C09145=1170.053,255.374,-66.162,-177.310,7.479,148.636
C09146=1170.048,255.622,-66.190,-177.307,7.482,148.635
C09147=1170.043,255.871,-66.218,-177.305,7.485,148.635
C09148=1170.039,256.120,-66.245,-177.302,7.488,148.635
C09149=1170.034,256.368,-66.273,-177.300,7.490,148.635
C09150=1170.030,256.617,-66.300,-177.297,7.493,148.635
C09151=1170.025,256.865,-66.328,-177.294,7.496,148.635
C09152=1170.021,257.114,-66.355,-177.291,7.499,148.635
C09153=1170.017,257.362,-66.383,-177.289,7.501,148.635
C09154=1170.012,257.610,-66.410,-177.286,7.504,148.635
C09155=1170.009,257.859,-66.438,-177.283,7.507,148.635
C09156=1170.004,258.107,-66.465,-177.280,7.510,148.635
C09157=1170.000,258.355,-66.493,-177.278,7.512,148.634
C09158=1169.996,258.604,-66.521,-177.276,7.515,148.634
C09159=1169.991,258.852,-66.548,-177.273,7.518,148.634
C09160=1169.987,259.101,-66.575,-177.270,7.521,148.634
C09161=1169.982,259.350,-66.604,-177.267,7.523,148.634
C09162=1169.977,259.598,-66.631,-177.265,7.526,148.634
C09163=1169.973,259.846,-66.659,-177.262,7.529,148.634
C09164=1169.969,260.095,-66.686,-177.259,7.532,148.634
C09165=1169.965,260.343,-66.714,-177.257,7.534,148.634
C09166=1169.960,260.591,-66.742,-177.254,7.537,148.634
C09167=1169.955,260.840,-66.770,-177.251,7.540,148.634
C09168=1169.951,261.088,-66.798,-177.249,7.543,148.634
C09169=1169.947,261.337,-66.826,-177.246,7.545,148.633
C09170=1169.943,261.585,-66.853,-177.244,7.548,148.633
C09171=1169.938,261.859,-66.884,-177.241,7.551,148.633
C09172=1169.933,262.131,-66.914,-177.238,7.553,148.633
C09173=1169.928,262.405,-66.945,-177.234,7.557,148.633
C09174=1169.924,262.677,-66.976,-177.232,7.560,148.633
C09175=1169.919,262.926,-67.003,-177.230,7.562,148.633
C09176=1169.915,263.175,-67.032,-177.227,7.565,148.633
C09177=1169.910,263.423,-67.060,-177.224,7.568,148.633
C09178=1169.907,263.671,-67.088,-177.221,7.571,148.633
C09179=1169.902,263.920,-67.115,-177.219,7.574,148.633
C09180=1169.897,264.168,-67.143,-177.216,7.576,148.633
C09181=1169.893,264.416,-67.171,-177.214,7.579,148.633
C09182=1169.889,264.664,-67.199,-177.211,7.582,148.633
C09183=1169.884,264.913,-67.228,-177.208,7.585,148.632
C09184=1169.880,265.161,-67.256,-177.205,7.588,148.632
C09185=1169.876,265.410,-67.283,-177.203,7.590,148.632
C09186=1169.871,265.658,-67.311,-177.200,7.593,148.632
C09187=1169.867,265.907,-67.340,-177.198,7.596,148.632
C09188=1169.863,266.155,-67.367,-177.195,7.599,148.632
C09189=1169.858,266.404,-67.396,-177.193,7.601,148.632
C09190=1169.854,266.652,-67.424,-177.190,7.604,148.632
C09191=1169.849,266.901,-67.453,-177.187,7.607,148.632
C09192=1169.845,267.148,-67.480,-177.184,7.610,148.632
C09193=1169.841,267.397,-67.509,-177.182,7.613,148.632
C09194=1169.836,267.645,-67.537,-177.180,7.615,148.632
C09195=1169.832,267.894,-67.565,-177.177,7.618,148.632
C09196=1169.827,268.142,-67.593,-177.174,7.621,148.632
C09197=1169.824,268.390,-67.622,-177.171,7.624,148.632
C09198=1169.818,268.639,-67.650,-177.169,7.627,148.632
C09199=1169.815,268.887,-67.678,-177.166,7.630,148.632
C09200=1169.810,269.135,-67.706,-177.164,7.632,148.631
C09201=1169.806,269.384,-67.735,-177.161,7.635,148.631
C09202=1169.801,269.632,-67.763,-177.158,7.638,148.631
C09203=1169.797,269.881,-67.791,-177.155,7.641,148.631
C09204=1169.792,270.128,-67.820,-177.153,7.644,148.631
C09205=1169.788,270.377,-67.848,-177.150,7.646,148.631
C09206=1169.784,270.626,-67.877,-177.148,7.649,148.631
C09207=1169.780,270.874,-67.905,-177.145,7.652,148.631
C09208=1169.775,271.123,-67.934,-177.142,7.655,148.631
C09209=1169.771,271.370,-67.961,-177.139,7.658,148.631
C09210=1169.767,271.619,-67.991,-177.137,7.661,148.631
C09211=1169.762,271.867,-68.019,-177.135,7.663,148.631
C09212=1169.758,272.115,-68.047,-177.132,7.666,148.631
C09213=1169.754,272.364,-68.075,-177.129,7.669,148.631
C09214=1169.749,272.612,-68.104,-177.126,7.672,148.631
C09215=1169.745,272.861,-68.133,-177.124,7.675,148.631
C09216=1169.741,273.109,-68.161,-177.121,7.678,148.631
C09217=1169.736,273.357,-68.190,-177.119,7.680,148.631
C09218=1169.732,273.605,-68.219,-177.116,7.683,148.631
C09219=1169.727,273.853,-68.247,-177.113,7.686,148.630
C09220=1169.723,274.102,-68.276,-177.110,7.689,148.630
C09221=1169.719,274.350,-68.305,-177.108,7.692,148.630
C09222=1169.714,274.598,-68.333,-177.105,7.695,148.631
C09223=1169.710,274.847,-68.362,-177.103,7.698,148.630
C09224=1169.706,275.095,-68.391,-177.100,7.701,148.630
C09225=1169.701,275.343,-68.419,-177.098,7.703,148.630
C09226=1169.697,275.592,-68.448,-177.095,7.706,148.630
C09227=1169.693,275.840,-68.477,-177.092,7.709,148.630
C09228=1169.688,276.089,-68.505,-177.089,7.712,148.630
C09229=1169.684,276.337,-68.534,-177.087,7.715,148.630
C09230=1169.680,276.585,-68.563,-177.085,7.718,148.630
C09231=1169.676,276.834,-68.592,-177.082,7.720,148.630
C09232=1169.671,277.082,-68.620,-177.079,7.723,148.630
C09233=1169.667,277.330,-68.650,-177.076,7.726,148.630
C09234=1169.663,277.579,-68.678,-177.074,7.730,148.630
C09235=1169.658,277.826,-68.707,-177.071,7.733,148.630
C09236=1169.654,278.075,-68.736,-177.069,7.736,148.630
C09237=1169.650,278.323,-68.765,-177.066,7.739,148.630
C09238=1169.646,278.571,-68.794,-177.064,7.741,148.630
C09239=1169.641,278.820,-68.822,-177.061,7.744,148.630
C09240=1169.637,279.068,-68.852,-177.058,7.747,148.630
C09241=1169.633,279.317,-68.881,-177.055,7.750,148.630
C09242=1169.628,279.565,-68.910,-177.053,7.753,148.630
C09243=1169.624,279.812,-68.939,-177.050,7.756,148.630
C09244=1169.620,280.061,-68.967,-177.048,7.759,148.630
C09245=1169.616,280.309,-68.997,-177.045,7.762,148.630
C09246=1169.611,280.558,-69.026,-177.043,7.764,148.630
C09247=1169.607,280.807,-69.055,-177.040,7.767,148.630
C09248=1169.602,281.054,-69.084,-177.037,7.770,148.630
C09249=1169.598,281.302,-69.114,-177.034,7.773,148.630
C09250=1169.594,281.551,-69.142,-177.032,7.776,148.630
C09251=1169.590,281.799,-69.171,-177.029,7.779,148.630
C09252=1169.586,282.047,-69.201,-177.027,7.782,148.630
C09253=1169.581,282.295,-69.230,-177.024,7.785,148.630
C09254=1169.577,282.544,-69.258,-177.022,7.787,148.630
C09255=1169.572,282.792,-69.288,-177.019,7.790,148.630
C09256=1169.568,283.040,-69.317,-177.016,7.793,148.630
C09257=1169.564,283.289,-69.347,-177.014,7.797,148.630
C09258=1169.560,283.537,-69.376,-177.011,7.799,148.630
C09259=1169.555,283.785,-69.405,-177.008,7.802,148.630
C09260=1169.551,284.033,-69.434,-177.006,7.805,148.630
C09261=1169.546,284.282,-69.464,-177.003,7.808,148.630
C09262=1169.542,284.530,-69.493,-177.000,7.811,148.630
C09263=1169.538,284.778,-69.522,-176.998,7.815,148.630
C09264=1169.534,285.026,-69.552,-176.996,7.817,148.630
C09265=1169.530,285.275,-69.581,-176.993,7.820,148.630
C09266=1169.525,285.522,-69.610,-176.990,7.823,148.630
C09267=1169.521,285.771,-69.640,-176.988,7.826,148.630
C09268=1169.517,286.019,-69.669,-176.985,7.829,148.630
C09269=1169.512,286.267,-69.699,-176.983,7.832,148.630
C09270=1169.508,286.515,-69.728,-176.980,7.835,148.630
C09271=1169.504,286.764,-69.758,-176.977,7.838,148.630
C09272=1169.500,287.012,-69.787,-176.974,7.841,148.630
C09273=1169.496,287.260,-69.817,-176.972,7.844,148.630
C09274=1169.491,287.508,-69.846,-176.969,7.847,148.630
C09275=1169.486,287.783,-69.878,-176.967,7.850,148.630
C09276=1169.481,288.058,-69.912,-176.964,7.853,148.630
C09277=1169.476,288.333,-69.944,-176.960,7.857,148.630
C09278=1169.472,288.608,-69.977,-176.958,7.860,148.630
C09279=1169.468,288.856,-70.007,-176.955,7.863,148.630
C09280=1169.463,289.105,-70.036,-176.953,7.866,148.630
C09281=1169.459,289.353,-70.066,-176.950,7.869,148.630
C09282=1169.455,289.601,-70.095,-176.947,7.872,148.630
C09283=1169.451,289.849,-70.125,-176.944,7.875,148.630
C09284=1169.447,290.098,-70.154,-176.942,7.878,148.630
C09285=1169.442,290.346,-70.185,-176.939,7.881,148.630
C09286=1169.438,290.594,-70.214,-176.937,7.883,148.630
C09287=1169.434,290.842,-70.244,-176.935,7.886,148.630
C09288=1169.429,291.090,-70.273,-176.932,7.890,148.630
C09289=1169.426,291.338,-70.304,-176.929,7.893,148.630
C09290=1169.421,291.587,-70.334,-176.927,7.896,148.630
C09291=1169.416,291.835,-70.363,-176.924,7.899,148.630
C09292=1169.412,292.083,-70.392,-176.922,7.902,148.630
C09293=1169.408,292.331,-70.423,-176.919,7.905,148.630
C09294=1169.404,292.579,-70.453,-176.916,7.908,148.630
C09295=1169.399,292.828,-70.482,-176.913,7.911,148.630
C09296=1169.395,293.075,-70.512,-176.911,7.914,148.630
C09297=1169.391,293.324,-70.542,-176.908,7.917,148.630
C09298=1169.386,293.572,-70.572,-176.906,7.920,148.630
C09299=1169.382,293.820,-70.602,-176.903,7.923,148.630
C09300=1169.378,294.068,-70.631,-176.901,7.926,148.630
C09301=1169.374,294.316,-70.662,-176.898,7.929,148.630
C09302=1169.370,294.564,-70.692,-176.895,7.932,148.630
C09303=1169.365,294.813,-70.721,-176.893,7.936,148.630
C09304=1169.361,295.061,-70.752,-176.890,7.939,148.630
C09305=1169.357,295.310,-70.782,-176.887,7.942,148.630
C09306=1169.353,295.557,-70.812,-176.885,7.944,148.630
C09307=1169.348,295.806,-70.842,-176.883,7.947,148.630
C09308=1169.344,296.053,-70.872,-176.880,7.950,148.630
C09309=1169.340,296.302,-70.902,-176.878,7.953,148.630
C09310=1169.336,296.550,-70.932,-176.875,7.956,148.630
C09311=1169.331,296.798,-70.962,-176.872,7.959,148.630
C09312=1169.327,297.046,-70.993,-176.870,7.962,148.630
C09313=1169.323,297.293,-71.023,-176.867,7.965,148.630
C09314=1169.319,297.543,-71.053,-176.865,7.968,148.630
C09315=1169.315,297.790,-71.083,-176.862,7.971,148.630
C09316=1169.311,298.039,-71.113,-176.859,7.974,148.630
C09317=1169.306,298.287,-71.143,-176.857,7.978,148.631
C09318=1169.302,298.534,-71.174,-176.854,7.981,148.631
C09319=1169.297,298.783,-71.204,-176.851,7.984,148.631
C09320=1169.294,299.031,-71.234,-176.849,7.987,148.631
C09321=1169.289,299.279,-71.265,-176.846,7.990,148.631
C09322=1169.285,299.527,-71.294,-176.844,7.993,148.631
C09323=1169.281,299.775,-71.325,-176.841,7.996,148.631
C09324=1169.277,300.023,-71.355,-176.839,7.999,148.631
C09325=1169.272,300.272,-71.385,-176.836,8.002,148.631
C09326=1169.268,300.520,-71.416,-176.834,8.005,148.631
C09327=1169.264,300.768,-71.447,-176.831,8.008,148.631
C09328=1169.259,301.016,-71.478,-176.829,8.012,148.631
C09329=1169.255,301.264,-71.507,-176.826,8.015,148.631
C09330=1169.250,301.512,-71.538,-176.823,8.018,148.631
C09331=1169.247,301.760,-71.568,-176.821,8.021,148.631
C09332=1169.243,302.008,-71.599,-176.818,8.024,148.631
C09333=1169.238,302.256,-71.630,-176.815,8.027,148.631
C09334=1169.234,302.504,-71.660,-176.813,8.030,148.631
C09335=1169.230,302.753,-71.690,-176.810,8.033,148.631
C09336=1169.226,303.001,-71.721,-176.808,8.036,148.631
C09337=1169.221,303.249,-71.751,-176.805,8.039,148.632
C09338=1169.217,303.497,-71.782,-176.803,8.042,148.632
C09339=1169.213,303.745,-71.813,-176.800,8.046,148.632
C09340=1169.209,303.993,-71.843,-176.798,8.049,148.632
C09341=1169.204,304.241,-71.874,-176.795,8.052,148.632
C09342=1169.200,304.489,-71.904,-176.793,8.055,148.632
C09343=1169.196,304.737,-71.935,-176.790,8.058,148.632
C09344=1169.192,304.985,-71.966,-176.787,8.061,148.632
C09345=1169.187,305.233,-71.997,-176.785,8.064,148.632
C09346=1169.184,305.482,-72.027,-176.782,8.067,148.632
C09347=1169.179,305.730,-72.058,-176.780,8.070,148.632
C09348=1169.175,305.978,-72.089,-176.777,8.073,148.632
C09349=1169.171,306.225,-72.119,-176.774,8.076,148.632
C09350=1169.167,306.474,-72.150,-176.772,8.080,148.632
C09351=1169.162,306.722,-72.181,-176.769,8.083,148.632
C09352=1169.157,306.970,-72.212,-176.767,8.086,148.632
C09353=1169.153,307.218,-72.243,-176.764,8.089,148.632
C09354=1169.150,307.466,-72.273,-176.762,8.092,148.633
C09355=1169.145,307.714,-72.304,-176.759,8.095,148.633
C09356=1169.141,307.962,-72.336,-176.756,8.098,148.633
C09357=1169.137,308.210,-72.367,-176.754,8.102,148.633
C09358=1169.132,308.458,-72.397,-176.751,8.105,148.633
C09359=1169.129,308.706,-72.428,-176.749,8.108,148.633
C09360=1169.124,308.954,-72.459,-176.746,8.111,148.633
C09361=1169.120,309.203,-72.490,-176.744,8.114,148.633
C09362=1169.116,309.450,-72.521,-176.741,8.118,148.633
C09363=1169.111,309.698,-72.552,-176.738,8.121,148.633
C09364=1169.107,309.947,-72.583,-176.736,8.124,148.633
C09365=1169.103,310.195,-72.613,-176.733,8.127,148.633
C09366=1169.100,310.443,-72.645,-176.731,8.130,148.633
C09367=1169.095,310.691,-72.676,-176.728,8.133,148.633
C09368=1169.090,310.939,-72.707,-176.726,8.137,148.634
C09369=1169.087,311.187,-72.738,-176.723,8.140,148.634
C09370=1169.082,311.435,-72.769,-176.721,8.143,148.634
C09371=1169.078,311.683,-72.800,-176.718,8.146,148.634
C09372=1169.074,311.931,-72.832,-176.716,8.149,148.634
C09373=1169.069,312.179,-72.863,-176.713,8.152,148.634
C09374=1169.065,312.427,-72.894,-176.711,8.156,148.634
C09375=1169.061,312.674,-72.925,-176.708,8.159,148.634
C09376=1169.057,312.923,-72.956,-176.706,8.162,148.634
C09377=1169.052,313.170,-72.988,-176.703,8.165,148.634
C09378=1169.048,313.419,-73.019,-176.701,8.168,148.635
C09379=1169.044,313.696,-73.054,-176.697,8.172,148.635
C09380=1169.039,313.972,-73.089,-176.695,8.175,148.635
C09381=1169.034,314.250,-73.123,-176.692,8.179,148.635
C09382=1169.030,314.526,-73.158,-176.689,8.182,148.635
C09383=1169.026,314.774,-73.190,-176.687,8.185,148.635
C09384=1169.021,315.023,-73.221,-176.683,8.189,148.635
C09385=1169.017,315.271,-73.253,-176.681,8.192,148.635
C09386=1169.013,315.519,-73.284,-176.678,8.195,148.635
C09387=1169.009,315.767,-73.316,-176.676,8.199,148.635
C09388=1169.004,316.015,-73.346,-176.673,8.202,148.635
C09389=1169.001,316.263,-73.378,-176.671,8.205,148.636
C09390=1168.997,316.511,-73.410,-176.668,8.208,148.636
C09391=1168.992,316.759,-73.441,-176.666,8.211,148.636
C09392=1168.989,317.007,-73.473,-176.664,8.214,148.636
C09393=1168.984,317.255,-73.503,-176.661,8.217,148.636
C09394=1168.980,317.503,-73.535,-176.659,8.221,148.636
C09395=1168.976,317.750,-73.567,-176.656,8.224,148.636
C09396=1168.971,317.998,-73.599,-176.654,8.227,148.636
C09397=1168.967,318.246,-73.630,-176.650,8.231,148.636
C09398=1168.963,318.494,-73.662,-176.648,8.234,148.637
C09399=1168.959,318.743,-73.694,-176.645,8.237,148.636
C09400=1168.955,318.990,-73.724,-176.643,8.240,148.637
C09401=1168.951,319.239,-73.756,-176.641,8.244,148.637
C09402=1168.946,319.486,-73.788,-176.638,8.247,148.637
C09403=1168.942,319.734,-73.820,-176.636,8.250,148.637
C09404=1168.939,319.982,-73.852,-176.633,8.253,148.637
C09405=1168.934,320.230,-73.883,-176.631,8.256,148.637
C09406=1168.930,320.478,-73.915,-176.628,8.259,148.637
C09407=1168.925,320.726,-73.947,-176.626,8.263,148.637
C09408=1168.922,320.974,-73.979,-176.623,8.266,148.638
C09409=1168.918,321.222,-74.010,-176.620,8.270,148.638
C09410=1168.914,321.469,-74.042,-176.618,8.273,148.638
C09411=1168.909,321.718,-74.074,-176.615,8.276,148.638
C09412=1168.905,321.966,-74.106,-176.613,8.279,148.638
C09413=1168.901,322.214,-74.137,-176.611,8.282,148.638
C09414=1168.896,322.462,-74.169,-176.608,8.285,148.638
C09415=1168.893,322.710,-74.201,-176.606,8.289,148.638
C09416=1168.888,322.957,-74.233,-176.603,8.292,148.638
C09417=1168.885,323.205,-74.265,-176.601,8.295,148.639
C09418=1168.880,323.454,-74.297,-176.598,8.299,148.639
C09419=1168.876,323.701,-74.329,-176.595,8.302,148.639
C09420=1168.872,323.949,-74.360,-176.593,8.305,148.639
C09421=1168.868,324.198,-74.393,-176.590,8.309,148.639
C09422=1168.863,324.445,-74.424,-176.588,8.312,148.639
C09423=1168.860,324.693,-74.456,-176.585,8.315,148.639
C09424=1168.855,324.941,-74.489,-176.583,8.318,148.639
C09425=1168.852,325.189,-74.521,-176.580,8.321,148.640
C09426=1168.847,325.436,-74.553,-176.578,8.325,148.640
C09427=1168.843,325.684,-74.585,-176.575,8.328,148.640
C09428=1168.839,325.932,-74.617,-176.572,8.332,148.640
C09429=1168.835,326.181,-74.649,-176.570,8.335,148.640
C09430=1168.831,326.428,-74.681,-176.567,8.338,148.640
C09431=1168.826,326.676,-74.713,-176.565,8.341,148.640
C09432=1168.823,326.924,-74.746,-176.563,8.345,148.641
C09433=1168.818,327.172,-74.778,-176.560,8.348,148.641
C09434=1168.814,327.420,-74.810,-176.558,8.351,148.641
C09435=1168.810,327.668,-74.842,-176.555,8.355,148.641
C09436=1168.806,327.916,-74.874,-176.552,8.358,148.641
C09437=1168.802,328.164,-74.907,-176.550,8.361,148.641
C09438=1168.797,328.411,-74.939,-176.548,8.365,148.642
C09439=1168.793,328.659,-74.971,-176.545,8.368,148.642
C09440=1168.789,328.907,-75.003,-176.543,8.371,148.642
C09441=1168.785,329.155,-75.036,-176.540,8.374,148.642
C09442=1168.781,329.403,-75.068,-176.537,8.378,148.642
C09443=1168.776,329.651,-75.100,-176.535,8.381,148.642
C09444=1168.773,329.898,-75.133,-176.532,8.384,148.642
C09445=1168.769,330.147,-75.165,-176.530,8.388,148.643
C09446=1168.765,330.395,-75.197,-176.528,8.391,148.643
C09447=1168.761,330.642,-75.230,-176.525,8.394,148.643
C09448=1168.756,330.890,-75.262,-176.523,8.397,148.643
C09449=1168.752,331.137,-75.295,-176.520,8.401,148.643
C09450=1168.748,331.386,-75.327,-176.517,8.404,148.643
C09451=1168.744,331.633,-75.360,-176.515,8.408,148.643
C09452=1168.740,331.881,-75.392,-176.513,8.411,148.644
C09453=1168.736,332.130,-75.425,-176.510,8.414,148.644
C09454=1168.732,332.377,-75.457,-176.508,8.418,148.644
C09455=1168.727,332.625,-75.489,-176.505,8.421,148.644
C09456=1168.723,332.873,-75.522,-176.503,8.425,148.644
C09457=1168.719,333.121,-75.554,-176.500,8.428,148.644
C09458=1168.715,333.368,-75.587,-176.498,8.431,148.645
C09459=1168.711,333.616,-75.620,-176.495,8.434,148.645
C09460=1168.707,333.864,-75.652,-176.493,8.438,148.645
C09461=1168.703,334.112,-75.685,-176.490,8.442,148.645
C09462=1168.699,334.360,-75.718,-176.488,8.445,148.645
C09463=1168.695,334.608,-75.751,-176.486,8.448,148.646
C09464=1168.691,334.855,-75.783,-176.483,8.451,148.646
C09465=1168.686,335.103,-75.816,-176.480,8.455,148.646
C09466=1168.682,335.351,-75.849,-176.478,8.458,148.646
C09467=1168.678,335.599,-75.881,-176.475,8.462,148.646
C09468=1168.674,335.847,-75.914,-176.473,8.465,148.646
C09469=1168.670,336.094,-75.947,-176.470,8.468,148.646
C09470=1168.666,336.342,-75.980,-176.468,8.472,148.647
C09471=1168.661,336.590,-76.013,-176.466,8.475,148.647
C09472=1168.658,336.838,-76.045,-176.463,8.479,148.647
C09473=1168.654,337.086,-76.078,-176.461,8.482,148.647
C09474=1168.649,337.334,-76.111,-176.458,8.486,148.647
C09475=1168.645,337.582,-76.144,-176.456,8.489,148.647
C09476=1168.641,337.829,-76.177,-176.453,8.492,148.648
C09477=1168.638,338.077,-76.210,-176.451,8.495,148.648
C09478=1168.634,338.324,-76.243,-176.448,8.499,148.648
C09479=1168.629,338.573,-76.275,-176.446,8.503,148.648
C09480=1168.625,338.821,-76.308,-176.444,8.506,148.649
C09481=1168.621,339.068,-76.342,-176.441,8.509,148.649
C09482=1168.617,339.316,-76.375,-176.439,8.513,148.649
C09483=1168.612,339.596,-76.412,-176.436,8.516,148.649
C09484=1168.608,339.874,-76.449,-176.433,8.520,148.649
C09485=1168.603,340.154,-76.486,-176.430,8.525,148.650
C09486=1168.598,340.433,-76.524,-176.428,8.528,148.650
C09487=1168.594,340.682,-76.556,-176.425,8.532,148.650
C09488=1168.590,340.929,-76.589,-176.423,8.535,148.650
C09489=1168.586,341.177,-76.623,-176.420,8.539,148.650
C09490=1168.582,341.425,-76.656,-176.418,8.542,148.651
C09491=1168.578,341.673,-76.689,-176.415,8.546,148.651
C09492=1168.573,341.920,-76.722,-176.413,8.549,148.651
C09493=1168.569,342.168,-76.755,-176.411,8.553,148.651
C09494=1168.565,342.416,-76.788,-176.408,8.556,148.651
C09495=1168.561,342.663,-76.822,-176.406,8.559,148.652
C09496=1168.558,342.911,-76.856,-176.403,8.563,148.652
C09497=1168.554,343.159,-76.889,-176.400,8.566,148.652
C09498=1168.549,343.407,-76.922,-176.398,8.570,148.652
C09499=1168.545,343.654,-76.955,-176.396,8.573,148.652
C09500=1168.541,343.902,-76.988,-176.393,8.577,148.653
C09501=1168.537,344.150,-77.022,-176.391,8.580,148.653
C09502=1168.533,344.398,-77.055,-176.388,8.584,148.653
C09503=1168.529,344.645,-77.088,-176.386,8.587,148.653
C09504=1168.525,344.893,-77.122,-176.384,8.590,148.654
C09505=1168.521,345.140,-77.155,-176.381,8.594,148.654
C09506=1168.517,345.389,-77.188,-176.379,8.598,148.654
C09507=1168.512,345.637,-77.222,-176.376,8.601,148.654
C09508=1168.508,345.884,-77.255,-176.374,8.604,148.654
C09509=1168.504,346.132,-77.289,-176.371,8.608,148.655
C09510=1168.500,346.379,-77.322,-176.369,8.612,148.655
C09511=1168.496,346.627,-77.356,-176.367,8.615,148.655
C09512=1168.492,346.875,-77.389,-176.364,8.618,148.655
C09513=1168.489,347.123,-77.423,-176.361,8.622,148.656
C09514=1168.484,347.371,-77.457,-176.360,8.626,148.656
C09515=1168.480,347.618,-77.490,-176.357,8.629,148.656
C09516=1168.476,347.865,-77.524,-176.355,8.633,148.656
C09517=1168.472,348.113,-77.557,-176.352,8.637,148.657
C09518=1168.468,348.362,-77.590,-176.350,8.640,148.657
C09519=1168.464,348.609,-77.625,-176.348,8.643,148.657
C09520=1168.460,348.857,-77.658,-176.345,8.647,148.657
C09521=1168.456,349.104,-77.692,-176.342,8.651,148.658
C09522=1168.452,349.352,-77.725,-176.340,8.654,148.658
C09523=1168.448,349.600,-77.759,-176.338,8.657,148.658
C09524=1168.443,349.847,-77.793,-176.335,8.661,148.658
C09525=1168.439,350.095,-77.826,-176.333,8.665,148.659
C09526=1168.435,350.342,-77.860,-176.331,8.668,148.659
C09527=1168.431,350.590,-77.894,-176.329,8.672,148.659
C09528=1168.427,350.838,-77.928,-176.326,8.676,148.659
C09529=1168.423,351.086,-77.961,-176.323,8.679,148.660
C09530=1168.419,351.333,-77.995,-176.321,8.682,148.660
C09531=1168.415,351.582,-78.029,-176.318,8.686,148.660
C09532=1168.411,351.829,-78.063,-176.316,8.690,148.660
C09533=1168.407,352.076,-78.097,-176.314,8.693,148.661
C09534=1168.403,352.324,-78.131,-176.312,8.697,148.661
C09535=1168.399,352.572,-78.165,-176.309,8.701,148.661
C09536=1168.395,352.819,-78.198,-176.307,8.704,148.661
C09537=1168.391,353.067,-78.233,-176.304,8.707,148.662
C09538=1168.387,353.315,-78.267,-176.302,8.712,148.662
C09539=1168.383,353.563,-78.301,-176.300,8.715,148.662
C09540=1168.379,353.810,-78.334,-176.297,8.718,148.663
C09541=1168.375,354.057,-78.368,-176.295,8.722,148.663
C09542=1168.371,354.306,-78.402,-176.292,8.726,148.663
C09543=1168.367,354.553,-78.436,-176.290,8.729,148.663
C09544=1168.362,354.800,-78.471,-176.288,8.733,148.664
C09545=1168.359,355.048,-78.505,-176.285,8.737,148.664
C09546=1168.355,355.296,-78.538,-176.283,8.740,148.664
C09547=1168.350,355.543,-78.573,-176.281,8.744,148.665
C09548=1168.347,355.791,-78.607,-176.278,8.748,148.665
C09549=1168.342,356.038,-78.641,-176.276,8.751,148.665
C09550=1168.339,356.286,-78.676,-176.274,8.755,148.666
C09551=1168.334,356.534,-78.709,-176.271,8.759,148.666
C09552=1168.331,356.781,-78.743,-176.269,8.762,148.666
C09553=1168.327,357.030,-78.778,-176.267,8.765,148.666
C09554=1168.323,357.277,-78.812,-176.264,8.770,148.667
C09555=1168.318,357.524,-78.846,-176.262,8.773,148.667
C09556=1168.315,357.772,-78.881,-176.260,8.776,148.667
C09557=1168.310,358.019,-78.915,-176.257,8.781,148.668
C09558=1168.307,358.267,-78.949,-176.255,8.784,148.668
C09559=1168.303,358.514,-78.984,-176.253,8.787,148.668
C09560=1168.299,358.763,-79.017,-176.250,8.792,148.669
C09561=1168.294,359.010,-79.052,-176.248,8.795,148.669
C09562=1168.291,359.257,-79.086,-176.246,8.798,148.669
C09563=1168.287,359.506,-79.120,-176.243,8.803,148.669
C09564=1168.282,359.753,-79.155,-176.241,8.806,148.670
C09565=1168.279,360.001,-79.189,-176.239,8.810,148.670
C09566=1168.274,360.248,-79.224,-176.236,8.814,148.670
C09567=1168.271,360.495,-79.259,-176.234,8.817,148.671
C09568=1168.267,360.743,-79.293,-176.232,8.821,148.671
C09569=1168.263,360.991,-79.328,-176.229,8.825,148.671
C09570=1168.259,361.238,-79.362,-176.227,8.829,148.672
C09571=1168.255,361.486,-79.397,-176.225,8.833,148.672
C09572=1168.250,361.734,-79.431,-176.223,8.836,148.672
C09573=1168.247,361.981,-79.465,-176.220,8.840,148.673
C09574=1168.243,362.229,-79.500,-176.218,8.844,148.673
C09575=1168.239,362.477,-79.535,-176.216,8.847,148.673
C09576=1168.235,362.723,-79.569,-176.214,8.851,148.674
C09577=1168.231,362.972,-79.604,-176.211,8.855,148.674
C09578=1168.227,363.219,-79.638,-176.209,8.859,148.674
C09579=1168.223,363.467,-79.673,-176.207,8.862,148.675
C09580=1168.219,363.714,-79.707,-176.204,8.866,148.675
C09581=1168.215,363.962,-79.743,-176.203,8.870,148.676
C09582=1168.211,364.209,-79.777,-176.201,8.874,148.676
C09583=1168.207,364.457,-79.811,-176.198,8.877,148.676
C09584=1168.203,364.704,-79.847,-176.196,8.881,148.677
C09585=1168.199,364.952,-79.881,-176.194,8.885,148.677
C09586=1168.195,365.199,-79.915,-176.192,8.888,148.678
C09587=1168.191,365.481,-79.955,-176.189,8.893,148.678
C09588=1168.186,365.764,-79.995,-176.187,8.897,148.678
C09589=1168.182,366.046,-80.035,-176.185,8.901,148.679
C09590=1168.177,366.328,-80.075,-176.182,8.906,148.679
C09591=1168.174,366.576,-80.109,-176.180,8.909,148.680
C09592=1168.169,366.823,-80.144,-176.178,8.913,148.680
C09593=1168.165,367.071,-80.179,-176.176,8.918,148.681
C09594=1168.161,367.319,-80.214,-176.174,8.921,148.681
C09595=1168.157,367.566,-80.249,-176.172,8.925,148.681
C09596=1168.153,367.814,-80.284,-176.171,8.928,148.682
C09597=1168.149,368.061,-80.319,-176.168,8.933,148.682
C09598=1168.146,368.308,-80.353,-176.166,8.936,148.683
C09599=1168.142,368.556,-80.389,-176.164,8.940,148.683
C09600=1168.137,368.803,-80.423,-176.163,8.944,148.684
C09601=1168.134,369.051,-80.459,-176.161,8.947,148.684
C09602=1168.130,369.299,-80.494,-176.159,8.951,148.684
C09603=1168.126,369.546,-80.529,-176.156,8.955,148.685
C09604=1168.122,369.794,-80.564,-176.155,8.959,148.685
C09605=1168.117,370.041,-80.599,-176.153,8.963,148.686
C09606=1168.113,370.289,-80.634,-176.151,8.966,148.686
C09607=1168.110,370.536,-80.669,-176.149,8.970,148.687
C09608=1168.105,370.783,-80.704,-176.148,8.974,148.687
C09609=1168.101,371.031,-80.739,-176.146,8.977,148.688
C09610=1168.098,371.279,-80.775,-176.144,8.981,148.688
C09611=1168.094,371.525,-80.810,-176.142,8.985,148.689
C09612=1168.090,371.774,-80.845,-176.141,8.989,148.689
C09613=1168.086,372.021,-80.880,-176.139,8.993,148.690
C09614=1168.082,372.268,-80.916,-176.137,8.997,148.690
C09615=1168.078,372.516,-80.950,-176.135,9.000,148.691
C09616=1168.074,372.764,-80.986,-176.133,9.004,148.691
C09617=1168.070,373.011,-81.021,-176.132,9.008,148.692
C09618=1168.066,373.258,-81.056,-176.130,9.012,148.692
C09619=1168.062,373.506,-81.092,-176.129,9.015,148.693
C09620=1168.058,373.753,-81.127,-176.128,9.019,148.694
C09621=1168.054,374.000,-81.162,-176.126,9.022,148.694
C09622=1168.050,374.248,-81.197,-176.125,9.026,148.695
C09623=1168.047,374.496,-81.233,-176.123,9.030,148.695
C09624=1168.043,374.743,-81.268,-176.121,9.034,148.696
C09625=1168.039,374.990,-81.303,-176.120,9.038,148.696
C09626=1168.035,375.238,-81.339,-176.119,9.041,148.697
C09627=1168.031,375.486,-81.374,-176.117,9.045,148.697
C09628=1168.027,375.733,-81.409,-176.116,9.048,148.698
C09629=1168.023,375.980,-81.444,-176.114,9.052,148.699
C09630=1168.019,376.228,-81.480,-176.113,9.056,148.699
C09631=1168.015,376.475,-81.516,-176.112,9.060,148.700
C09632=1168.011,376.723,-81.552,-176.110,9.064,148.700
C09633=1168.007,376.970,-81.587,-176.109,9.067,148.701
C09634=1168.003,377.217,-81.622,-176.108,9.071,148.702
C09635=1167.999,377.465,-81.657,-176.106,9.075,148.702
C09636=1167.996,377.713,-81.693,-176.106,9.078,148.703
C09637=1167.992,377.960,-81.728,-176.104,9.082,148.704
C09638=1167.987,378.207,-81.764,-176.103,9.086,148.704
C09639=1167.983,378.455,-81.800,-176.102,9.089,148.705
C09640=1167.980,378.702,-81.835,-176.100,9.093,148.705
C09641=1167.976,378.950,-81.871,-176.100,9.096,148.706
C09642=1167.972,379.197,-81.906,-176.098,9.100,148.707
C09643=1167.967,379.445,-81.942,-176.097,9.104,148.707
C09644=1167.964,379.692,-81.978,-176.096,9.107,148.708
C09645=1167.960,379.940,-82.013,-176.095,9.111,148.709
C09646=1167.956,380.187,-82.049,-176.094,9.114,148.709
C09647=1167.952,380.434,-82.084,-176.093,9.118,148.710
C09648=1167.948,380.682,-82.120,-176.092,9.121,148.711
C09649=1167.944,380.929,-82.156,-176.091,9.124,148.711
C09650=1167.940,381.177,-82.191,-176.090,9.128,148.712
C09651=1167.937,381.424,-82.227,-176.090,9.132,148.713
C09652=1167.932,381.671,-82.263,-176.089,9.135,148.713
C09653=1167.928,381.918,-82.299,-176.088,9.139,148.714
C09654=1167.925,382.166,-82.334,-176.087,9.142,148.715
C09655=1167.921,382.413,-82.370,-176.086,9.145,148.715
C09656=1167.917,382.661,-82.406,-176.085,9.150,148.716
C09657=1167.913,382.908,-82.442,-176.085,9.153,148.717
C09658=1167.909,383.156,-82.477,-176.084,9.156,148.717
C09659=1167.904,383.403,-82.513,-176.083,9.159,148.718
C09660=1167.901,383.650,-82.549,-176.083,9.162,148.719
C09661=1167.897,383.897,-82.585,-176.082,9.166,148.720
C09662=1167.894,384.145,-82.620,-176.081,9.170,148.720
C09663=1167.889,384.393,-82.656,-176.081,9.173,148.721
C09664=1167.886,384.640,-82.692,-176.080,9.177,148.722
C09665=1167.882,384.888,-82.727,-176.080,9.180,148.723
C09666=1167.877,385.134,-82.764,-176.079,9.183,148.723
C09667=1167.874,385.382,-82.799,-176.078,9.186,148.724
C09668=1167.870,385.629,-82.835,-176.078,9.190,148.725
C09669=1167.866,385.877,-82.871,-176.078,9.193,148.725
C09670=1167.862,386.124,-82.907,-176.078,9.196,148.726
C09671=1167.859,386.371,-82.943,-176.077,9.199,148.727
C09672=1167.854,386.619,-82.979,-176.077,9.202,148.727
C09673=1167.850,386.867,-83.015,-176.076,9.206,148.728
C09674=1167.847,387.114,-83.050,-176.076,9.209,148.729
C09675=1167.842,387.361,-83.087,-176.076,9.212,148.730
C09676=1167.838,387.608,-83.122,-176.075,9.215,148.730
C09677=1167.834,387.856,-83.158,-176.075,9.218,148.731
C09678=1167.831,388.103,-83.195,-176.075,9.221,148.732
C09679=1167.827,388.350,-83.230,-176.075,9.224,148.733
C09680=1167.823,388.598,-83.266,-176.074,9.228,148.734
C09681=1167.819,388.845,-83.303,-176.074,9.230,148.734
C09682=1167.816,389.093,-83.338,-176.074,9.234,148.735
C09683=1167.811,389.340,-83.374,-176.074,9.236,148.736
C09684=1167.808,389.588,-83.410,-176.074,9.240,148.736
C09685=1167.803,389.835,-83.447,-176.074,9.242,148.737
C09686=1167.800,390.083,-83.482,-176.074,9.245,148.738
C09687=1167.796,390.329,-83.517,-176.074,9.248,148.739
C09688=1167.791,390.577,-83.554,-176.074,9.251,148.740
C09689=1167.788,390.824,-83.590,-176.074,9.254,148.740
C09690=1167.784,391.071,-83.627,-176.074,9.257,148.741
C09691=1167.779,391.357,-83.668,-176.074,9.261,148.742
C09692=1167.775,391.642,-83.709,-176.074,9.263,148.743
C09693=1167.771,391.927,-83.751,-176.074,9.267,148.744
C09694=1167.766,392.212,-83.792,-176.074,9.270,148.744
C09695=1167.762,392.459,-83.829,-176.075,9.272,148.745
C09696=1167.758,392.707,-83.865,-176.074,9.276,148.746
C09697=1167.755,392.954,-83.901,-176.074,9.278,148.747
C09698=1167.751,393.201,-83.937,-176.075,9.281,148.748
C09699=1167.747,393.449,-83.973,-176.075,9.284,148.748
C09700=1167.743,393.696,-84.009,-176.075,9.286,148.749
C09701=1167.739,393.944,-84.045,-176.075,9.289,148.750
C09702=1167.735,394.191,-84.081,-176.076,9.292,148.751
C09703=1167.731,394.438,-84.117,-176.076,9.294,148.751
C09704=1167.727,394.686,-84.153,-176.076,9.297,148.752
C09705=1167.723,394.933,-84.190,-176.076,9.299,148.753
C09706=1167.719,395.180,-84.225,-176.076,9.302,148.753
C09707=1167.715,395.427,-84.262,-176.076,9.304,148.754
C09708=1167.711,395.675,-84.297,-176.077,9.307,148.755
C09709=1167.708,395.922,-84.334,-176.077,9.310,148.756
C09710=1167.704,396.169,-84.370,-176.077,9.312,148.756
C09711=1167.700,396.417,-84.405,-176.077,9.315,148.757
C09712=1167.696,396.664,-84.442,-176.078,9.317,148.758
C09713=1167.692,396.912,-84.478,-176.078,9.319,148.759
C09714=1167.688,397.159,-84.515,-176.078,9.322,148.759
C09715=1167.684,397.406,-84.550,-176.079,9.325,148.760
C09716=1167.680,397.653,-84.587,-176.079,9.327,148.761
C09717=1167.677,397.901,-84.623,-176.080,9.329,148.762
C09718=1167.672,398.148,-84.659,-176.080,9.332,148.762
C09719=1167.669,398.396,-84.695,-176.080,9.334,148.763
C09720=1167.665,398.643,-84.732,-176.081,9.336,148.764
C09721=1167.661,398.890,-84.767,-176.081,9.338,148.764
C09722=1167.657,399.137,-84.804,-176.081,9.341,148.765
C09723=1167.653,399.385,-84.840,-176.081,9.344,148.766
C09724=1167.649,399.632,-84.877,-176.082,9.345,148.766
C09725=1167.646,399.880,-84.912,-176.082,9.348,148.767
C09726=1167.641,400.127,-84.949,-176.083,9.350,148.768
C09727=1167.638,400.374,-84.985,-176.083,9.353,148.769
C09728=1167.634,400.622,-85.022,-176.084,9.355,148.769
C09729=1167.630,400.869,-85.057,-176.084,9.357,148.770
C09730=1167.626,401.116,-85.094,-176.084,9.359,148.771
C09731=1167.622,401.364,-85.129,-176.085,9.361,148.771
C09732=1167.618,401.611,-85.166,-176.085,9.364,148.772
C09733=1167.615,401.858,-85.202,-176.086,9.365,148.773
C09734=1167.610,402.106,-85.239,-176.086,9.368,148.773
C09735=1167.606,402.353,-85.275,-176.087,9.370,148.774
C09736=1167.603,402.600,-85.311,-176.087,9.372,148.775
C09737=1167.598,402.848,-85.347,-176.088,9.374,148.776
C09738=1167.595,403.095,-85.384,-176.088,9.377,148.776
C09739=1167.591,403.343,-85.420,-176.088,9.378,148.777
C09740=1167.587,403.590,-85.456,-176.088,9.381,148.777
C09741=1167.583,403.838,-85.492,-176.089,9.382,148.778
C09742=1167.579,404.084,-85.528,-176.089,9.385,148.779
C09743=1167.575,404.332,-85.564,-176.090,9.387,148.779
C09744=1167.572,404.579,-85.601,-176.090,9.389,148.780
C09745=1167.568,404.826,-85.638,-176.091,9.391,148.781
C09746=1167.564,405.074,-85.673,-176.091,9.393,148.781
C09747=1167.560,405.321,-85.710,-176.091,9.395,148.782
C09748=1167.556,405.568,-85.746,-176.092,9.397,148.783
C09749=1167.552,405.816,-85.782,-176.092,9.399,148.783
C09750=1167.548,406.063,-85.819,-176.093,9.401,148.784
C09751=1167.544,406.310,-85.855,-176.093,9.403,148.785
C09752=1167.540,406.558,-85.891,-176.093,9.405,148.785
C09753=1167.537,406.805,-85.927,-176.094,9.407,148.786
C09754=1167.532,407.052,-85.964,-176.094,9.409,148.786
C09755=1167.529,407.300,-86.000,-176.095,9.411,148.787
C09756=1167.525,407.547,-86.037,-176.095,9.413,148.788
C09757=1167.521,407.794,-86.072,-176.096,9.415,148.788
C09758=1167.517,408.042,-86.109,-176.096,9.417,148.789
C09759=1167.513,408.289,-86.146,-176.096,9.419,148.790
C09760=1167.509,408.536,-86.181,-176.097,9.420,148.790
C09761=1167.505,408.783,-86.218,-176.097,9.423,148.791
C09762=1167.501,409.031,-86.254,-176.098,9.424,148.791
C09763=1167.497,409.278,-86.291,-176.098,9.426,148.792
C09764=1167.494,409.526,-86.326,-176.099,9.428,148.793
C09765=1167.490,409.773,-86.363,-176.099,9.430,148.793
C09766=1167.486,410.020,-86.399,-176.099,9.432,148.794
C09767=1167.482,410.268,-86.435,-176.100,9.434,148.795
C09768=1167.478,410.515,-86.472,-176.100,9.436,148.795
C09769=1167.474,410.762,-86.508,-176.101,9.438,148.796
C09770=1167.470,411.009,-86.545,-176.101,9.439,148.796
C09771=1167.467,411.256,-86.581,-176.102,9.441,148.797
C09772=1167.462,411.504,-86.617,-176.102,9.443,148.797
C09773=1167.459,411.751,-86.653,-176.102,9.445,148.798
C09774=1167.455,411.998,-86.690,-176.103,9.447,148.799
C09775=1167.450,412.246,-86.726,-176.103,9.448,148.799
C09776=1167.447,412.493,-86.763,-176.103,9.451,148.800
C09777=1167.443,412.741,-86.799,-176.104,9.452,148.800
C09778=1167.439,412.988,-86.835,-176.104,9.454,148.801
C09779=1167.435,413.235,-86.872,-176.105,9.456,148.802
C09780=1167.431,413.483,-86.908,-176.104,9.458,148.802
C09781=1167.427,413.729,-86.944,-176.105,9.460,148.803
C09782=1167.423,413.977,-86.980,-176.105,9.461,148.803
C09783=1167.420,414.224,-87.017,-176.106,9.463,148.804
C09784=1167.416,414.471,-87.054,-176.106,9.465,148.804
C09785=1167.411,414.719,-87.090,-176.107,9.467,148.805
C09786=1167.408,414.966,-87.126,-176.107,9.468,148.805
C09787=1167.404,415.213,-87.163,-176.108,9.470,148.806
C09788=1167.401,415.461,-87.199,-176.108,9.471,148.806
C09789=1167.398,415.709,-87.235,-176.108,9.474,148.807
C09790=1167.397,415.955,-87.271,-176.108,9.475,148.808
C09791=1167.396,416.263,-87.316,-176.109,9.477,148.808
C09792=1167.397,416.570,-87.360,-176.109,9.479,148.809
C09793=1167.399,416.877,-87.405,-176.109,9.481,148.809
C09794=1167.403,417.184,-87.449,-176.109,9.484,148.810
C09795=1166.981,417.185,-87.494,-176.113,9.495,148.814
C09796=1166.978,416.875,-87.450,-176.113,9.492,148.813
C09797=1166.976,416.565,-87.405,-176.112,9.490,148.813
C09798=1166.975,416.255,-87.360,-176.112,9.488,148.812
C09799=1166.975,415.945,-87.315,-176.111,9.486,148.811
C09800=1166.977,415.697,-87.279,-176.111,9.485,148.811
C09801=1166.980,415.449,-87.242,-176.111,9.482,148.810
C09802=1166.983,415.202,-87.206,-176.110,9.481,148.810
C09803=1166.987,414.955,-87.170,-176.110,9.479,148.809
C09804=1166.991,414.708,-87.133,-176.109,9.477,148.808
C09805=1166.995,414.461,-87.096,-176.109,9.476,148.808
C09806=1166.999,414.213,-87.061,-176.109,9.473,148.807
C09807=1167.003,413.966,-87.024,-176.109,9.472,148.807
C09808=1167.006,413.719,-86.988,-176.108,9.470,148.806
C09809=1167.010,413.471,-86.952,-176.108,9.469,148.806
C09810=1167.014,413.224,-86.915,-176.108,9.466,148.805
C09811=1167.018,412.976,-86.879,-176.107,9.465,148.805
C09812=1167.022,412.729,-86.842,-176.107,9.463,148.804
C09813=1167.026,412.482,-86.806,-176.106,9.461,148.803
C09814=1167.030,412.235,-86.770,-176.106,9.459,148.803
C09815=1167.034,411.987,-86.733,-176.105,9.457,148.802
C09816=1167.037,411.741,-86.697,-176.105,9.456,148.802
C09817=1167.042,411.493,-86.661,-176.104,9.454,148.801
C09818=1167.045,411.246,-86.624,-176.104,9.452,148.800
C09819=1167.050,410.998,-86.588,-176.104,9.450,148.800
C09820=1167.054,410.751,-86.551,-176.103,9.448,148.799
C09821=1167.057,410.504,-86.515,-176.103,9.447,148.799
C09822=1167.061,410.255,-86.479,-176.103,9.444,148.798
C09823=1167.064,410.009,-86.442,-176.102,9.443,148.797
C09824=1167.068,409.761,-86.405,-176.102,9.441,148.797
C09825=1167.072,409.514,-86.370,-176.101,9.439,148.796
C09826=1167.076,409.267,-86.333,-176.101,9.437,148.796
C09827=1167.080,409.019,-86.297,-176.100,9.435,148.795
C09828=1167.084,408.772,-86.261,-176.100,9.434,148.795
C09829=1167.088,408.525,-86.224,-176.100,9.431,148.794
C09830=1167.092,408.277,-86.188,-176.099,9.429,148.793
C09831=1167.096,408.030,-86.151,-176.099,9.428,148.793
C09832=1167.099,407.783,-86.116,-176.098,9.426,148.792
C09833=1167.103,407.535,-86.079,-176.098,9.424,148.791
C09834=1167.107,407.289,-86.043,-176.097,9.422,148.791
C09835=1167.111,407.041,-86.007,-176.097,9.420,148.790
C09836=1167.115,406.794,-85.970,-176.097,9.418,148.790
C09837=1167.119,406.546,-85.934,-176.096,9.416,148.789
C09838=1167.123,406.299,-85.897,-176.096,9.414,148.788
C09839=1167.127,406.051,-85.862,-176.095,9.412,148.788
C09840=1167.131,405.804,-85.825,-176.095,9.410,148.787
C09841=1167.134,405.557,-85.789,-176.094,9.408,148.786
C09842=1167.139,405.309,-85.752,-176.094,9.406,148.786
C09843=1167.142,405.063,-85.716,-176.094,9.404,148.785
C09844=1167.146,404.815,-85.680,-176.093,9.402,148.784
C09845=1167.150,404.568,-85.643,-176.093,9.400,148.784
C09846=1167.154,404.320,-85.608,-176.092,9.398,148.783
C09847=1167.158,404.073,-85.571,-176.092,9.396,148.782
C09848=1167.162,403.826,-85.535,-176.091,9.394,148.782
C09849=1167.166,403.578,-85.498,-176.091,9.391,148.781
C09850=1167.169,403.331,-85.462,-176.090,9.390,148.780
C09851=1167.174,403.083,-85.426,-176.090,9.387,148.780
C09852=1167.177,402.837,-85.390,-176.089,9.385,148.779
C09853=1167.181,402.589,-85.354,-176.089,9.383,148.778
C09854=1167.185,402.342,-85.317,-176.089,9.381,148.778
C09855=1167.189,402.094,-85.281,-176.088,9.379,148.777
C09856=1167.193,401.847,-85.245,-176.088,9.377,148.776
C09857=1167.197,401.599,-85.209,-176.088,9.374,148.776
C09858=1167.200,401.353,-85.173,-176.087,9.372,148.775
C09859=1167.205,401.105,-85.136,-176.087,9.370,148.774
C09860=1167.209,400.858,-85.100,-176.086,9.368,148.773
C09861=1167.212,400.610,-85.064,-176.086,9.365,148.773
C09862=1167.217,400.363,-85.027,-176.085,9.364,148.772
C09863=1167.220,400.116,-84.991,-176.085,9.361,148.771
C09864=1167.224,399.868,-84.955,-176.084,9.359,148.771
C09865=1167.228,399.621,-84.918,-176.084,9.357,148.770
C09866=1167.232,399.373,-84.882,-176.084,9.354,148.769
C09867=1167.235,399.127,-84.846,-176.083,9.353,148.769
C09868=1167.240,398.879,-84.810,-176.083,9.350,148.768
C09869=1167.243,398.632,-84.774,-176.083,9.347,148.767
C09870=1167.248,398.384,-84.737,-176.082,9.346,148.767
C09871=1167.251,398.137,-84.701,-176.082,9.343,148.766
C09872=1167.255,397.889,-84.665,-176.082,9.340,148.765
C09873=1167.259,397.642,-84.630,-176.082,9.338,148.764
C09874=1167.263,397.395,-84.593,-176.081,9.336,148.764
C09875=1167.267,397.147,-84.557,-176.081,9.333,148.763
C09876=1167.271,396.900,-84.520,-176.081,9.331,148.762
C09877=1167.275,396.653,-84.485,-176.080,9.328,148.761
C09878=1167.279,396.406,-84.448,-176.080,9.325,148.761
C09879=1167.283,396.159,-84.413,-176.079,9.324,148.760
C09880=1167.287,395.911,-84.376,-176.079,9.321,148.759
C09881=1167.291,395.664,-84.340,-176.079,9.318,148.759
C09882=1167.295,395.417,-84.303,-176.079,9.316,148.758
C09883=1167.298,395.169,-84.268,-176.079,9.313,148.757
C09884=1167.302,394.922,-84.231,-176.078,9.310,148.756
C09885=1167.306,394.674,-84.195,-176.078,9.308,148.755
C09886=1167.310,394.427,-84.160,-176.078,9.305,148.755
C09887=1167.314,394.180,-84.123,-176.078,9.303,148.754
C09888=1167.318,393.932,-84.088,-176.077,9.300,148.753
C09889=1167.322,393.685,-84.051,-176.077,9.297,148.752
C09890=1167.325,393.438,-84.015,-176.077,9.295,148.752
C09891=1167.329,393.190,-83.978,-176.077,9.292,148.751
C09892=1167.333,392.943,-83.943,-176.076,9.290,148.750
C09893=1167.337,392.695,-83.907,-176.076,9.287,148.750
C09894=1167.341,392.448,-83.870,-176.076,9.284,148.749
C09895=1167.345,392.200,-83.834,-176.076,9.281,148.748
C09896=1167.350,391.916,-83.792,-176.076,9.278,148.747
C09897=1167.354,391.630,-83.751,-176.076,9.274,148.746
C09898=1167.359,391.346,-83.709,-176.076,9.272,148.745
C09899=1167.363,391.060,-83.668,-176.076,9.268,148.745
C09900=1167.367,390.813,-83.632,-176.076,9.266,148.744
C09901=1167.371,390.565,-83.595,-176.076,9.262,148.743
C09902=1167.375,390.319,-83.560,-176.075,9.259,148.742
C09903=1167.379,390.071,-83.525,-176.075,9.257,148.741
C09904=1167.383,389.824,-83.488,-176.076,9.253,148.741
C09905=1167.386,389.576,-83.452,-176.076,9.251,148.740
C09906=1167.390,389.329,-83.415,-176.076,9.247,148.739
C09907=1167.394,389.082,-83.380,-176.076,9.245,148.738
C09908=1167.398,388.834,-83.344,-176.076,9.241,148.738
C09909=1167.402,388.586,-83.308,-176.076,9.239,148.737
C09910=1167.406,388.340,-83.272,-176.077,9.236,148.736
C09911=1167.410,388.092,-83.236,-176.076,9.233,148.735
C09912=1167.414,387.844,-83.200,-176.077,9.230,148.735
C09913=1167.417,387.597,-83.164,-176.077,9.226,148.734
C09914=1167.421,387.350,-83.128,-176.077,9.224,148.733
C09915=1167.426,387.103,-83.093,-176.078,9.220,148.732
C09916=1167.429,386.856,-83.056,-176.078,9.217,148.732
C09917=1167.433,386.608,-83.020,-176.078,9.213,148.731
C09918=1167.437,386.361,-82.985,-176.079,9.210,148.730
C09919=1167.441,386.113,-82.949,-176.079,9.207,148.729
C09920=1167.445,385.866,-82.912,-176.079,9.204,148.729
C09921=1167.448,385.618,-82.877,-176.080,9.201,148.728
C09922=1167.452,385.371,-82.841,-176.080,9.198,148.727
C09923=1167.456,385.123,-82.805,-176.081,9.194,148.727
C09924=1167.460,384.876,-82.769,-176.081,9.191,148.726
C09925=1167.464,384.629,-82.734,-176.082,9.187,148.725
C09926=1167.469,384.382,-82.698,-176.083,9.184,148.724
C09927=1167.472,384.134,-82.662,-176.083,9.181,148.724
C09928=1167.476,383.887,-82.626,-176.083,9.178,148.723
C09929=1167.480,383.639,-82.590,-176.084,9.174,148.722
C09930=1167.484,383.392,-82.554,-176.085,9.170,148.721
C09931=1167.487,383.144,-82.518,-176.086,9.167,148.721
C09932=1167.492,382.897,-82.483,-176.086,9.164,148.720
C09933=1167.496,382.650,-82.447,-176.087,9.160,148.719
C09934=1167.500,382.402,-82.412,-176.088,9.156,148.719
C09935=1167.503,382.155,-82.376,-176.089,9.153,148.718
C09936=1167.508,381.907,-82.340,-176.089,9.150,148.717
C09937=1167.511,381.660,-82.304,-176.090,9.147,148.717
C09938=1167.515,381.413,-82.268,-176.091,9.142,148.716
C09939=1167.519,381.166,-82.233,-176.092,9.139,148.715
C09940=1167.523,380.918,-82.197,-176.093,9.135,148.715
C09941=1167.527,380.670,-82.161,-176.094,9.132,148.714
C09942=1167.531,380.423,-82.126,-176.095,9.129,148.713
C09943=1167.534,380.175,-82.090,-176.096,9.125,148.713
C09944=1167.539,379.928,-82.054,-176.096,9.122,148.712
C09945=1167.543,379.681,-82.019,-176.098,9.118,148.711
C09946=1167.547,379.433,-81.983,-176.099,9.115,148.711
C09947=1167.550,379.186,-81.948,-176.100,9.111,148.710
C09948=1167.555,378.938,-81.912,-176.101,9.107,148.709
C09949=1167.558,378.690,-81.876,-176.102,9.103,148.709
C09950=1167.563,378.444,-81.841,-176.103,9.100,148.708
C09951=1167.566,378.196,-81.805,-176.104,9.096,148.707
C09952=1167.570,377.949,-81.770,-176.106,9.093,148.707
C09953=1167.574,377.701,-81.734,-176.107,9.089,148.706
C09954=1167.579,377.454,-81.698,-176.108,9.086,148.706
C09955=1167.582,377.207,-81.663,-176.109,9.082,148.705
C09956=1167.586,376.959,-81.627,-176.111,9.078,148.704
C09957=1167.590,376.712,-81.592,-176.112,9.074,148.704
C09958=1167.593,376.464,-81.556,-176.113,9.071,148.703
C09959=1167.598,376.217,-81.522,-176.114,9.067,148.703
C09960=1167.602,375.969,-81.486,-176.116,9.063,148.702
C09961=1167.606,375.721,-81.450,-176.117,9.059,148.701
C09962=1167.610,375.474,-81.415,-176.119,9.055,148.701
C09963=1167.614,375.227,-81.379,-176.120,9.052,148.700
C09964=1167.617,374.980,-81.344,-176.121,9.048,148.700
C09965=1167.621,374.732,-81.308,-176.123,9.045,148.699
C09966=1167.625,374.484,-81.273,-176.125,9.041,148.699
C09967=1167.629,374.237,-81.238,-176.126,9.037,148.698
C09968=1167.633,373.990,-81.203,-176.128,9.033,148.697
C09969=1167.637,373.742,-81.167,-176.129,9.030,148.697
C09970=1167.641,373.495,-81.132,-176.131,9.026,148.696
C09971=1167.645,373.247,-81.097,-176.133,9.022,148.696
C09972=1167.649,373.000,-81.062,-176.134,9.018,148.695
C09973=1167.652,372.752,-81.026,-176.136,9.014,148.695
C09974=1167.657,372.505,-80.992,-176.137,9.011,148.694
C09975=1167.661,372.257,-80.956,-176.139,9.007,148.694
C09976=1167.664,372.010,-80.920,-176.141,9.003,148.693
C09977=1167.668,371.763,-80.885,-176.143,8.999,148.693
C09978=1167.672,371.515,-80.850,-176.144,8.996,148.692
C09979=1167.676,371.267,-80.815,-176.146,8.992,148.692
C09980=1167.681,371.020,-80.780,-176.148,8.988,148.691
C09981=1167.684,370.772,-80.745,-176.150,8.985,148.691
C09982=1167.688,370.525,-80.709,-176.151,8.981,148.690
C09983=1167.693,370.278,-80.675,-176.153,8.977,148.690
C09984=1167.696,370.030,-80.639,-176.155,8.973,148.689
C09985=1167.700,369.783,-80.604,-176.157,8.969,148.689
C09986=1167.704,369.535,-80.569,-176.159,8.966,148.688
C09987=1167.708,369.288,-80.534,-176.160,8.962,148.688
C09988=1167.712,369.039,-80.499,-176.162,8.958,148.687
C09989=1167.716,368.793,-80.464,-176.164,8.954,148.687
C09990=1167.720,368.545,-80.429,-176.167,8.950,148.686
C09991=1167.725,368.298,-80.394,-176.168,8.946,148.686
C09992=1167.729,368.050,-80.359,-176.170,8.943,148.686
C09993=1167.731,367.802,-80.324,-176.172,8.939,148.685
C09994=1167.736,367.555,-80.289,-176.175,8.935,148.685
C09995=1167.740,367.308,-80.254,-176.176,8.931,148.684
C09996=1167.744,367.060,-80.219,-176.178,8.928,148.684
//INST
///DATE 2021/06/15 17:25
///ATTR SC,RW,RJ
////FRAME ROBOT
///GROUP1 RB1
NOP
MOVL C00000 V=800.0 PL=0
MOVL C00001 V=800.0 PL=0
MOVL C00002 V=800.0 PL=0
MOVL C00003 V=800.0 PL=0
MOVL C00004 V=800.0 PL=0
MOVL C00005 V=800.0 PL=0
MOVL C00006 V=800.0 PL=0
MOVL C00007 V=800.0 PL=0
MOVL C00008 V=800.0 PL=0
MOVL C00009 V=800.0 PL=0
MOVL C00010 V=800.0 PL=0
MOVL C00011 V=800.0 PL=0
MOVL C00012 V=800.0 PL=0
MOVL C00013 V=800.0 PL=0
MOVL C00014 V=800.0 PL=0
MOVL C00015 V=800.0 PL=0
MOVL C00016 V=800.0 PL=0
MOVL C00017 V=800.0 PL=0
MOVL C00018 V=800.0 PL=0
MOVL C00019 V=800.0 PL=0
MOVL C00020 V=800.0 PL=0
MOVL C00021 V=800.0 PL=0
MOVL C00022 V=800.0 PL=0
MOVL C00023 V=800.0 PL=0
MOVL C00024 V=800.0 PL=0
MOVL C00025 V=800.0 PL=0
MOVL C00026 V=800.0 PL=0
MOVL C00027 V=800.0 PL=0
MOVL C00028 V=800.0 PL=0
MOVL C00029 V=800.0 PL=0
MOVL C00030 V=800.0 PL=0
MOVL C00031 V=800.0 PL=0
MOVL C00032 V=800.0 PL=0
MOVL C00033 V=800.0 PL=0
MOVL C00034 V=800.0 PL=0
MOVL C00035 V=800.0 PL=0
MOVL C00036 V=800.0 PL=0
MOVL C00037 V=800.0 PL=0
MOVL C00038 V=800.0 PL=0
MOVL C00039 V=800.0 PL=0
MOVL C00040 V=800.0 PL=0
MOVL C00041 V=800.0 PL=0
MOVL C00042 V=800.0 PL=0
MOVL C00043 V=800.0 PL=0
MOVL C00044 V=800.0 PL=0
MOVL C00045 V=800.0 PL=0
MOVL C00046 V=800.0 PL=0
MOVL C00047 V=800.0 PL=0
MOVL C00048 V=800.0 PL=0
MOVL C00049 V=800.0 PL=0
MOVL C00050 V=800.0 PL=0
MOVL C00051 V=800.0 PL=0
MOVL C00052 V=800.0 PL=0
MOVL C00053 V=800.0 PL=0
MOVL C00054 V=800.0 PL=0
MOVL C00055 V=800.0 PL=0
MOVL C00056 V=800.0 PL=0
MOVL C00057 V=800.0 PL=0
MOVL C00058 V=800.0 PL=0
MOVL C00059 V=800.0 PL=0
MOVL C00060 V=800.0 PL=0
MOVL C00061 V=800.0 PL=0
MOVL C00062 V=800.0 PL=0
MOVL C00063 V=800.0 PL=0
MOVL C00064 V=800.0 PL=0
MOVL C00065 V=800.0 PL=0
MOVL C00066 V=800.0 PL=0
MOVL C00067 V=800.0 PL=0
MOVL C00068 V=800.0 PL=0
MOVL C00069 V=800.0 PL=0
MOVL C00070 V=800.0 PL=0
MOVL C00071 V=800.0 PL=0
MOVL C00072 V=800.0 PL=0
MOVL C00073 V=800.0 PL=0
MOVL C00074 V=800.0 PL=0
MOVL C00075 V=800.0 PL=0
MOVL C00076 V=800.0 PL=0
MOVL C00077 V=800.0 PL=0
MOVL C00078 V=800.0 PL=0
MOVL C00079 V=800.0 PL=0
MOVL C00080 V=800.0 PL=0
MOVL C00081 V=800.0 PL=0
MOVL C00082 V=800.0 PL=0
MOVL C00083 V=800.0 PL=0
MOVL C00084 V=800.0 PL=0
MOVL C00085 V=800.0 PL=0
MOVL C00086 V=800.0 PL=0
MOVL C00087 V=800.0 PL=0
MOVL C00088 V=800.0 PL=0
MOVL C00089 V=800.0 PL=0
MOVL C00090 V=800.0 PL=0
MOVL C00091 V=800.0 PL=0
MOVL C00092 V=800.0 PL=0
MOVL C00093 V=800.0 PL=0
MOVL C00094 V=800.0 PL=0
MOVL C00095 V=800.0 PL=0
MOVL C00096 V=800.0 PL=0
MOVL C00097 V=800.0 PL=0
MOVL C00098 V=800.0 PL=0
MOVL C00099 V=800.0 PL=0
MOVL C00100 V=800.0 PL=0
MOVL C00101 V=800.0 PL=0
MOVL C00102 V=800.0 PL=0
MOVL C00103 V=800.0 PL=0
MOVL C00104 V=800.0 PL=0
MOVL C00105 V=800.0 PL=0
MOVL C00106 V=800.0 PL=0
MOVL C00107 V=800.0 PL=0
MOVL C00108 V=800.0 PL=0
MOVL C00109 V=800.0 PL=0
MOVL C00110 V=800.0 PL=0
MOVL C00111 V=800.0 PL=0
MOVL C00112 V=800.0 PL=0
MOVL C00113 V=800.0 PL=0
MOVL C00114 V=800.0 PL=0
MOVL C00115 V=800.0 PL=0
MOVL C00116 V=800.0 PL=0
MOVL C00117 V=800.0 PL=0
MOVL C00118 V=800.0 PL=0
MOVL C00119 V=800.0 PL=0
MOVL C00120 V=800.0 PL=0
MOVL C00121 V=800.0 PL=0
MOVL C00122 V=800.0 PL=0
MOVL C00123 V=800.0 PL=0
MOVL C00124 V=800.0 PL=0
MOVL C00125 V=800.0 PL=0
MOVL C00126 V=800.0 PL=0
MOVL C00127 V=800.0 PL=0
MOVL C00128 V=800.0 PL=0
MOVL C00129 V=800.0 PL=0
MOVL C00130 V=800.0 PL=0
MOVL C00131 V=800.0 PL=0
MOVL C00132 V=800.0 PL=0
MOVL C00133 V=800.0 PL=0
MOVL C00134 V=800.0 PL=0
MOVL C00135 V=800.0 PL=0
MOVL C00136 V=800.0 PL=0
MOVL C00137 V=800.0 PL=0
MOVL C00138 V=800.0 PL=0
MOVL C00139 V=800.0 PL=0
MOVL C00140 V=800.0 PL=0
MOVL C00141 V=800.0 PL=0
MOVL C00142 V=800.0 PL=0
MOVL C00143 V=800.0 PL=0
MOVL C00144 V=800.0 PL=0
MOVL C00145 V=800.0 PL=0
MOVL C00146 V=800.0 PL=0
MOVL C00147 V=800.0 PL=0
MOVL C00148 V=800.0 PL=0
MOVL C00149 V=800.0 PL=0
MOVL C00150 V=800.0 PL=0
MOVL C00151 V=800.0 PL=0
MOVL C00152 V=800.0 PL=0
MOVL C00153 V=800.0 PL=0
MOVL C00154 V=800.0 PL=0
MOVL C00155 V=800.0 PL=0
MOVL C00156 V=800.0 PL=0
MOVL C00157 V=800.0 PL=0
MOVL C00158 V=800.0 PL=0
MOVL C00159 V=800.0 PL=0
MOVL C00160 V=800.0 PL=0
MOVL C00161 V=800.0 PL=0
MOVL C00162 V=800.0 PL=0
MOVL C00163 V=800.0 PL=0
MOVL C00164 V=800.0 PL=0
MOVL C00165 V=800.0 PL=0
MOVL C00166 V=800.0 PL=0
MOVL C00167 V=800.0 PL=0
MOVL C00168 V=800.0 PL=0
MOVL C00169 V=800.0 PL=0
MOVL C00170 V=800.0 PL=0
MOVL C00171 V=800.0 PL=0
MOVL C00172 V=800.0 PL=0
MOVL C00173 V=800.0 PL=0
MOVL C00174 V=800.0 PL=0
MOVL C00175 V=800.0 PL=0
MOVL C00176 V=800.0 PL=0
MOVL C00177 V=800.0 PL=0
MOVL C00178 V=800.0 PL=0
MOVL C00179 V=800.0 PL=0
MOVL C00180 V=800.0 PL=0
MOVL C00181 V=800.0 PL=0
MOVL C00182 V=800.0 PL=0
MOVL C00183 V=800.0 PL=0
MOVL C00184 V=800.0 PL=0
MOVL C00185 V=800.0 PL=0
MOVL C00186 V=800.0 PL=0
MOVL C00187 V=800.0 PL=0
MOVL C00188 V=800.0 PL=0
MOVL C00189 V=800.0 PL=0
MOVL C00190 V=800.0 PL=0
MOVL C00191 V=800.0 PL=0
MOVL C00192 V=800.0 PL=0
MOVL C00193 V=800.0 PL=0
MOVL C00194 V=800.0 PL=0
MOVL C00195 V=800.0 PL=0
MOVL C00196 V=800.0 PL=0
MOVL C00197 V=800.0 PL=0
MOVL C00198 V=800.0 PL=0
MOVL C00199 V=800.0 PL=0
MOVL C00200 V=800.0 PL=0
MOVL C00201 V=800.0 PL=0
MOVL C00202 V=800.0 PL=0
MOVL C00203 V=800.0 PL=0
MOVL C00204 V=800.0 PL=0
MOVL C00205 V=800.0 PL=0
MOVL C00206 V=800.0 PL=0
MOVL C00207 V=800.0 PL=0
MOVL C00208 V=800.0 PL=0
MOVL C00209 V=800.0 PL=0
MOVL C00210 V=800.0 PL=0
MOVL C00211 V=800.0 PL=0
MOVL C00212 V=800.0 PL=0
MOVL C00213 V=800.0 PL=0
MOVL C00214 V=800.0 PL=0
MOVL C00215 V=800.0 PL=0
MOVL C00216 V=800.0 PL=0
MOVL C00217 V=800.0 PL=0
MOVL C00218 V=800.0 PL=0
MOVL C00219 V=800.0 PL=0
MOVL C00220 V=800.0 PL=0
MOVL C00221 V=800.0 PL=0
MOVL C00222 V=800.0 PL=0
MOVL C00223 V=800.0 PL=0
MOVL C00224 V=800.0 PL=0
MOVL C00225 V=800.0 PL=0
MOVL C00226 V=800.0 PL=0
MOVL C00227 V=800.0 PL=0
MOVL C00228 V=800.0 PL=0
MOVL C00229 V=800.0 PL=0
MOVL C00230 V=800.0 PL=0
MOVL C00231 V=800.0 PL=0
MOVL C00232 V=800.0 PL=0
MOVL C00233 V=800.0 PL=0
MOVL C00234 V=800.0 PL=0
MOVL C00235 V=800.0 PL=0
MOVL C00236 V=800.0 PL=0
MOVL C00237 V=800.0 PL=0
MOVL C00238 V=800.0 PL=0
MOVL C00239 V=800.0 PL=0
MOVL C00240 V=800.0 PL=0
MOVL C00241 V=800.0 PL=0
MOVL C00242 V=800.0 PL=0
MOVL C00243 V=800.0 PL=0
MOVL C00244 V=800.0 PL=0
MOVL C00245 V=800.0 PL=0
MOVL C00246 V=800.0 PL=0
MOVL C00247 V=800.0 PL=0
MOVL C00248 V=800.0 PL=0
MOVL C00249 V=800.0 PL=0
MOVL C00250 V=800.0 PL=0
MOVL C00251 V=800.0 PL=0
MOVL C00252 V=800.0 PL=0
MOVL C00253 V=800.0 PL=0
MOVL C00254 V=800.0 PL=0
MOVL C00255 V=800.0 PL=0
MOVL C00256 V=800.0 PL=0
MOVL C00257 V=800.0 PL=0
MOVL C00258 V=800.0 PL=0
MOVL C00259 V=800.0 PL=0
MOVL C00260 V=800.0 PL=0
MOVL C00261 V=800.0 PL=0
MOVL C00262 V=800.0 PL=0
MOVL C00263 V=800.0 PL=0
MOVL C00264 V=800.0 PL=0
MOVL C00265 V=800.0 PL=0
MOVL C00266 V=800.0 PL=0
MOVL C00267 V=800.0 PL=0
MOVL C00268 V=800.0 PL=0
MOVL C00269 V=800.0 PL=0
MOVL C00270 V=800.0 PL=0
MOVL C00271 V=800.0 PL=0
MOVL C00272 V=800.0 PL=0
MOVL C00273 V=800.0 PL=0
MOVL C00274 V=800.0 PL=0
MOVL C00275 V=800.0 PL=0
MOVL C00276 V=800.0 PL=0
MOVL C00277 V=800.0 PL=0
MOVL C00278 V=800.0 PL=0
MOVL C00279 V=800.0 PL=0
MOVL C00280 V=800.0 PL=0
MOVL C00281 V=800.0 PL=0
MOVL C00282 V=800.0 PL=0
MOVL C00283 V=800.0 PL=0
MOVL C00284 V=800.0 PL=0
MOVL C00285 V=800.0 PL=0
MOVL C00286 V=800.0 PL=0
MOVL C00287 V=800.0 PL=0
MOVL C00288 V=800.0 PL=0
MOVL C00289 V=800.0 PL=0
MOVL C00290 V=800.0 PL=0
MOVL C00291 V=800.0 PL=0
MOVL C00292 V=800.0 PL=0
MOVL C00293 V=800.0 PL=0
MOVL C00294 V=800.0 PL=0
MOVL C00295 V=800.0 PL=0
MOVL C00296 V=800.0 PL=0
MOVL C00297 V=800.0 PL=0
MOVL C00298 V=800.0 PL=0
MOVL C00299 V=800.0 PL=0
MOVL C00300 V=800.0 PL=0
MOVL C00301 V=800.0 PL=0
MOVL C00302 V=800.0 PL=0
MOVL C00303 V=800.0 PL=0
MOVL C00304 V=800.0 PL=0
MOVL C00305 V=800.0 PL=0
MOVL C00306 V=800.0 PL=0
MOVL C00307 V=800.0 PL=0
MOVL C00308 V=800.0 PL=0
MOVL C00309 V=800.0 PL=0
MOVL C00310 V=800.0 PL=0
MOVL C00311 V=800.0 PL=0
MOVL C00312 V=800.0 PL=0
MOVL C00313 V=800.0 PL=0
MOVL C00314 V=800.0 PL=0
MOVL C00315 V=800.0 PL=0
MOVL C00316 V=800.0 PL=0
MOVL C00317 V=800.0 PL=0
MOVL C00318 V=800.0 PL=0
MOVL C00319 V=800.0 PL=0
MOVL C00320 V=800.0 PL=0
MOVL C00321 V=800.0 PL=0
MOVL C00322 V=800.0 PL=0
MOVL C00323 V=800.0 PL=0
MOVL C00324 V=800.0 PL=0
MOVL C00325 V=800.0 PL=0
MOVL C00326 V=800.0 PL=0
MOVL C00327 V=800.0 PL=0
MOVL C00328 V=800.0 PL=0
MOVL C00329 V=800.0 PL=0
MOVL C00330 V=800.0 PL=0
MOVL C00331 V=800.0 PL=0
MOVL C00332 V=800.0 PL=0
MOVL C00333 V=800.0 PL=0
MOVL C00334 V=800.0 PL=0
MOVL C00335 V=800.0 PL=0
MOVL C00336 V=800.0 PL=0
MOVL C00337 V=800.0 PL=0
MOVL C00338 V=800.0 PL=0
MOVL C00339 V=800.0 PL=0
MOVL C00340 V=800.0 PL=0
MOVL C00341 V=800.0 PL=0
MOVL C00342 V=800.0 PL=0
MOVL C00343 V=800.0 PL=0
MOVL C00344 V=800.0 PL=0
MOVL C00345 V=800.0 PL=0
MOVL C00346 V=800.0 PL=0
MOVL C00347 V=800.0 PL=0
MOVL C00348 V=800.0 PL=0
MOVL C00349 V=800.0 PL=0
MOVL C00350 V=800.0 PL=0
MOVL C00351 V=800.0 PL=0
MOVL C00352 V=800.0 PL=0
MOVL C00353 V=800.0 PL=0
MOVL C00354 V=800.0 PL=0
MOVL C00355 V=800.0 PL=0
MOVL C00356 V=800.0 PL=0
MOVL C00357 V=800.0 PL=0
MOVL C00358 V=800.0 PL=0
MOVL C00359 V=800.0 PL=0
MOVL C00360 V=800.0 PL=0
MOVL C00361 V=800.0 PL=0
MOVL C00362 V=800.0 PL=0
MOVL C00363 V=800.0 PL=0
MOVL C00364 V=800.0 PL=0
MOVL C00365 V=800.0 PL=0
MOVL C00366 V=800.0 PL=0
MOVL C00367 V=800.0 PL=0
MOVL C00368 V=800.0 PL=0
MOVL C00369 V=800.0 PL=0
MOVL C00370 V=800.0 PL=0
MOVL C00371 V=800.0 PL=0
MOVL C00372 V=800.0 PL=0
MOVL C00373 V=800.0 PL=0
MOVL C00374 V=800.0 PL=0
MOVL C00375 V=800.0 PL=0
MOVL C00376 V=800.0 PL=0
MOVL C00377 V=800.0 PL=0
MOVL C00378 V=800.0 PL=0
MOVL C00379 V=800.0 PL=0
MOVL C00380 V=800.0 PL=0
MOVL C00381 V=800.0 PL=0
MOVL C00382 V=800.0 PL=0
MOVL C00383 V=800.0 PL=0
MOVL C00384 V=800.0 PL=0
MOVL C00385 V=800.0 PL=0
MOVL C00386 V=800.0 PL=0
MOVL C00387 V=800.0 PL=0
MOVL C00388 V=800.0 PL=0
MOVL C00389 V=800.0 PL=0
MOVL C00390 V=800.0 PL=0
MOVL C00391 V=800.0 PL=0
MOVL C00392 V=800.0 PL=0
MOVL C00393 V=800.0 PL=0
MOVL C00394 V=800.0 PL=0
MOVL C00395 V=800.0 PL=0
MOVL C00396 V=800.0 PL=0
MOVL C00397 V=800.0 PL=0
MOVL C00398 V=800.0 PL=0
MOVL C00399 V=800.0 PL=0
MOVL C00400 V=800.0 PL=0
MOVL C00401 V=800.0 PL=0
MOVL C00402 V=800.0 PL=0
MOVL C00403 V=800.0 PL=0
MOVL C00404 V=800.0 PL=0
MOVL C00405 V=800.0 PL=0
MOVL C00406 V=800.0 PL=0
MOVL C00407 V=800.0 PL=0
MOVL C00408 V=800.0 PL=0
MOVL C00409 V=800.0 PL=0
MOVL C00410 V=800.0 PL=0
MOVL C00411 V=800.0 PL=0
MOVL C00412 V=800.0 PL=0
MOVL C00413 V=800.0 PL=0
MOVL C00414 V=800.0 PL=0
MOVL C00415 V=800.0 PL=0
MOVL C00416 V=800.0 PL=0
MOVL C00417 V=800.0 PL=0
MOVL C00418 V=800.0 PL=0
MOVL C00419 V=800.0 PL=0
MOVL C00420 V=800.0 PL=0
MOVL C00421 V=800.0 PL=0
MOVL C00422 V=800.0 PL=0
MOVL C00423 V=800.0 PL=0
MOVL C00424 V=800.0 PL=0
MOVL C00425 V=800.0 PL=0
MOVL C00426 V=800.0 PL=0
MOVL C00427 V=800.0 PL=0
MOVL C00428 V=800.0 PL=0
MOVL C00429 V=800.0 PL=0
MOVL C00430 V=800.0 PL=0
MOVL C00431 V=800.0 PL=0
MOVL C00432 V=800.0 PL=0
MOVL C00433 V=800.0 PL=0
MOVL C00434 V=800.0 PL=0
MOVL C00435 V=800.0 PL=0
MOVL C00436 V=800.0 PL=0
MOVL C00437 V=800.0 PL=0
MOVL C00438 V=800.0 PL=0
MOVL C00439 V=800.0 PL=0
MOVL C00440 V=800.0 PL=0
MOVL C00441 V=800.0 PL=0
MOVL C00442 V=800.0 PL=0
MOVL C00443 V=800.0 PL=0
MOVL C00444 V=800.0 PL=0
MOVL C00445 V=800.0 PL=0
MOVL C00446 V=800.0 PL=0
MOVL C00447 V=800.0 PL=0
MOVL C00448 V=800.0 PL=0
MOVL C00449 V=800.0 PL=0
MOVL C00450 V=800.0 PL=0
MOVL C00451 V=800.0 PL=0
MOVL C00452 V=800.0 PL=0
MOVL C00453 V=800.0 PL=0
MOVL C00454 V=800.0 PL=0
MOVL C00455 V=800.0 PL=0
MOVL C00456 V=800.0 PL=0
MOVL C00457 V=800.0 PL=0
MOVL C00458 V=800.0 PL=0
MOVL C00459 V=800.0 PL=0
MOVL C00460 V=800.0 PL=0
MOVL C00461 V=800.0 PL=0
MOVL C00462 V=800.0 PL=0
MOVL C00463 V=800.0 PL=0
MOVL C00464 V=800.0 PL=0
MOVL C00465 V=800.0 PL=0
MOVL C00466 V=800.0 PL=0
MOVL C00467 V=800.0 PL=0
MOVL C00468 V=800.0 PL=0
MOVL C00469 V=800.0 PL=0
MOVL C00470 V=800.0 PL=0
MOVL C00471 V=800.0 PL=0
MOVL C00472 V=800.0 PL=0
MOVL C00473 V=800.0 PL=0
MOVL C00474 V=800.0 PL=0
MOVL C00475 V=800.0 PL=0
MOVL C00476 V=800.0 PL=0
MOVL C00477 V=800.0 PL=0
MOVL C00478 V=800.0 PL=0
MOVL C00479 V=800.0 PL=0
MOVL C00480 V=800.0 PL=0
MOVL C00481 V=800.0 PL=0
MOVL C00482 V=800.0 PL=0
MOVL C00483 V=800.0 PL=0
MOVL C00484 V=800.0 PL=0
MOVL C00485 V=800.0 PL=0
MOVL C00486 V=800.0 PL=0
MOVL C00487 V=800.0 PL=0
MOVL C00488 V=800.0 PL=0
MOVL C00489 V=800.0 PL=0
MOVL C00490 V=800.0 PL=0
MOVL C00491 V=800.0 PL=0
MOVL C00492 V=800.0 PL=0
MOVL C00493 V=800.0 PL=0
MOVL C00494 V=800.0 PL=0
MOVL C00495 V=800.0 PL=0
MOVL C00496 V=800.0 PL=0
MOVL C00497 V=800.0 PL=0
MOVL C00498 V=800.0 PL=0
MOVL C00499 V=800.0 PL=0
MOVL C00500 V=800.0 PL=0
MOVL C00501 V=800.0 PL=0
MOVL C00502 V=800.0 PL=0
MOVL C00503 V=800.0 PL=0
MOVL C00504 V=800.0 PL=0
MOVL C00505 V=800.0 PL=0
MOVL C00506 V=800.0 PL=0
MOVL C00507 V=800.0 PL=0
MOVL C00508 V=800.0 PL=0
MOVL C00509 V=800.0 PL=0
MOVL C00510 V=800.0 PL=0
MOVL C00511 V=800.0 PL=0
MOVL C00512 V=800.0 PL=0
MOVL C00513 V=800.0 PL=0
MOVL C00514 V=800.0 PL=0
MOVL C00515 V=800.0 PL=0
MOVL C00516 V=800.0 PL=0
MOVL C00517 V=800.0 PL=0
MOVL C00518 V=800.0 PL=0
MOVL C00519 V=800.0 PL=0
MOVL C00520 V=800.0 PL=0
MOVL C00521 V=800.0 PL=0
MOVL C00522 V=800.0 PL=0
MOVL C00523 V=800.0 PL=0
MOVL C00524 V=800.0 PL=0
MOVL C00525 V=800.0 PL=0
MOVL C00526 V=800.0 PL=0
MOVL C00527 V=800.0 PL=0
MOVL C00528 V=800.0 PL=0
MOVL C00529 V=800.0 PL=0
MOVL C00530 V=800.0 PL=0
MOVL C00531 V=800.0 PL=0
MOVL C00532 V=800.0 PL=0
MOVL C00533 V=800.0 PL=0
MOVL C00534 V=800.0 PL=0
MOVL C00535 V=800.0 PL=0
MOVL C00536 V=800.0 PL=0
MOVL C00537 V=800.0 PL=0
MOVL C00538 V=800.0 PL=0
MOVL C00539 V=800.0 PL=0
MOVL C00540 V=800.0 PL=0
MOVL C00541 V=800.0 PL=0
MOVL C00542 V=800.0 PL=0
MOVL C00543 V=800.0 PL=0
MOVL C00544 V=800.0 PL=0
MOVL C00545 V=800.0 PL=0
MOVL C00546 V=800.0 PL=0
MOVL C00547 V=800.0 PL=0
MOVL C00548 V=800.0 PL=0
MOVL C00549 V=800.0 PL=0
MOVL C00550 V=800.0 PL=0
MOVL C00551 V=800.0 PL=0
MOVL C00552 V=800.0 PL=0
MOVL C00553 V=800.0 PL=0
MOVL C00554 V=800.0 PL=0
MOVL C00555 V=800.0 PL=0
MOVL C00556 V=800.0 PL=0
MOVL C00557 V=800.0 PL=0
MOVL C00558 V=800.0 PL=0
MOVL C00559 V=800.0 PL=0
MOVL C00560 V=800.0 PL=0
MOVL C00561 V=800.0 PL=0
MOVL C00562 V=800.0 PL=0
MOVL C00563 V=800.0 PL=0
MOVL C00564 V=800.0 PL=0
MOVL C00565 V=800.0 PL=0
MOVL C00566 V=800.0 PL=0
MOVL C00567 V=800.0 PL=0
MOVL C00568 V=800.0 PL=0
MOVL C00569 V=800.0 PL=0
MOVL C00570 V=800.0 PL=0
MOVL C00571 V=800.0 PL=0
MOVL C00572 V=800.0 PL=0
MOVL C00573 V=800.0 PL=0
MOVL C00574 V=800.0 PL=0
MOVL C00575 V=800.0 PL=0
MOVL C00576 V=800.0 PL=0
MOVL C00577 V=800.0 PL=0
MOVL C00578 V=800.0 PL=0
MOVL C00579 V=800.0 PL=0
MOVL C00580 V=800.0 PL=0
MOVL C00581 V=800.0 PL=0
MOVL C00582 V=800.0 PL=0
MOVL C00583 V=800.0 PL=0
MOVL C00584 V=800.0 PL=0
MOVL C00585 V=800.0 PL=0
MOVL C00586 V=800.0 PL=0
MOVL C00587 V=800.0 PL=0
MOVL C00588 V=800.0 PL=0
MOVL C00589 V=800.0 PL=0
MOVL C00590 V=800.0 PL=0
MOVL C00591 V=800.0 PL=0
MOVL C00592 V=800.0 PL=0
MOVL C00593 V=800.0 PL=0
MOVL C00594 V=800.0 PL=0
MOVL C00595 V=800.0 PL=0
MOVL C00596 V=800.0 PL=0
MOVL C00597 V=800.0 PL=0
MOVL C00598 V=800.0 PL=0
MOVL C00599 V=800.0 PL=0
MOVL C00600 V=800.0 PL=0
MOVL C00601 V=800.0 PL=0
MOVL C00602 V=800.0 PL=0
MOVL C00603 V=800.0 PL=0
MOVL C00604 V=800.0 PL=0
MOVL C00605 V=800.0 PL=0
MOVL C00606 V=800.0 PL=0
MOVL C00607 V=800.0 PL=0
MOVL C00608 V=800.0 PL=0
MOVL C00609 V=800.0 PL=0
MOVL C00610 V=800.0 PL=0
MOVL C00611 V=800.0 PL=0
MOVL C00612 V=800.0 PL=0
MOVL C00613 V=800.0 PL=0
MOVL C00614 V=800.0 PL=0
MOVL C00615 V=800.0 PL=0
MOVL C00616 V=800.0 PL=0
MOVL C00617 V=800.0 PL=0
MOVL C00618 V=800.0 PL=0
MOVL C00619 V=800.0 PL=0
MOVL C00620 V=800.0 PL=0
MOVL C00621 V=800.0 PL=0
MOVL C00622 V=800.0 PL=0
MOVL C00623 V=800.0 PL=0
MOVL C00624 V=800.0 PL=0
MOVL C00625 V=800.0 PL=0
MOVL C00626 V=800.0 PL=0
MOVL C00627 V=800.0 PL=0
MOVL C00628 V=800.0 PL=0
MOVL C00629 V=800.0 PL=0
MOVL C00630 V=800.0 PL=0
MOVL C00631 V=800.0 PL=0
MOVL C00632 V=800.0 PL=0
MOVL C00633 V=800.0 PL=0
MOVL C00634 V=800.0 PL=0
MOVL C00635 V=800.0 PL=0
MOVL C00636 V=800.0 PL=0
MOVL C00637 V=800.0 PL=0
MOVL C00638 V=800.0 PL=0
MOVL C00639 V=800.0 PL=0
MOVL C00640 V=800.0 PL=0
MOVL C00641 V=800.0 PL=0
MOVL C00642 V=800.0 PL=0
MOVL C00643 V=800.0 PL=0
MOVL C00644 V=800.0 PL=0
MOVL C00645 V=800.0 PL=0
MOVL C00646 V=800.0 PL=0
MOVL C00647 V=800.0 PL=0
MOVL C00648 V=800.0 PL=0
MOVL C00649 V=800.0 PL=0
MOVL C00650 V=800.0 PL=0
MOVL C00651 V=800.0 PL=0
MOVL C00652 V=800.0 PL=0
MOVL C00653 V=800.0 PL=0
MOVL C00654 V=800.0 PL=0
MOVL C00655 V=800.0 PL=0
MOVL C00656 V=800.0 PL=0
MOVL C00657 V=800.0 PL=0
MOVL C00658 V=800.0 PL=0
MOVL C00659 V=800.0 PL=0
MOVL C00660 V=800.0 PL=0
MOVL C00661 V=800.0 PL=0
MOVL C00662 V=800.0 PL=0
MOVL C00663 V=800.0 PL=0
MOVL C00664 V=800.0 PL=0
MOVL C00665 V=800.0 PL=0
MOVL C00666 V=800.0 PL=0
MOVL C00667 V=800.0 PL=0
MOVL C00668 V=800.0 PL=0
MOVL C00669 V=800.0 PL=0
MOVL C00670 V=800.0 PL=0
MOVL C00671 V=800.0 PL=0
MOVL C00672 V=800.0 PL=0
MOVL C00673 V=800.0 PL=0
MOVL C00674 V=800.0 PL=0
MOVL C00675 V=800.0 PL=0
MOVL C00676 V=800.0 PL=0
MOVL C00677 V=800.0 PL=0
MOVL C00678 V=800.0 PL=0
MOVL C00679 V=800.0 PL=0
MOVL C00680 V=800.0 PL=0
MOVL C00681 V=800.0 PL=0
MOVL C00682 V=800.0 PL=0
MOVL C00683 V=800.0 PL=0
MOVL C00684 V=800.0 PL=0
MOVL C00685 V=800.0 PL=0
MOVL C00686 V=800.0 PL=0
MOVL C00687 V=800.0 PL=0
MOVL C00688 V=800.0 PL=0
MOVL C00689 V=800.0 PL=0
MOVL C00690 V=800.0 PL=0
MOVL C00691 V=800.0 PL=0
MOVL C00692 V=800.0 PL=0
MOVL C00693 V=800.0 PL=0
MOVL C00694 V=800.0 PL=0
MOVL C00695 V=800.0 PL=0
MOVL C00696 V=800.0 PL=0
MOVL C00697 V=800.0 PL=0
MOVL C00698 V=800.0 PL=0
MOVL C00699 V=800.0 PL=0
MOVL C00700 V=800.0 PL=0
MOVL C00701 V=800.0 PL=0
MOVL C00702 V=800.0 PL=0
MOVL C00703 V=800.0 PL=0
MOVL C00704 V=800.0 PL=0
MOVL C00705 V=800.0 PL=0
MOVL C00706 V=800.0 PL=0
MOVL C00707 V=800.0 PL=0
MOVL C00708 V=800.0 PL=0
MOVL C00709 V=800.0 PL=0
MOVL C00710 V=800.0 PL=0
MOVL C00711 V=800.0 PL=0
MOVL C00712 V=800.0 PL=0
MOVL C00713 V=800.0 PL=0
MOVL C00714 V=800.0 PL=0
MOVL C00715 V=800.0 PL=0
MOVL C00716 V=800.0 PL=0
MOVL C00717 V=800.0 PL=0
MOVL C00718 V=800.0 PL=0
MOVL C00719 V=800.0 PL=0
MOVL C00720 V=800.0 PL=0
MOVL C00721 V=800.0 PL=0
MOVL C00722 V=800.0 PL=0
MOVL C00723 V=800.0 PL=0
MOVL C00724 V=800.0 PL=0
MOVL C00725 V=800.0 PL=0
MOVL C00726 V=800.0 PL=0
MOVL C00727 V=800.0 PL=0
MOVL C00728 V=800.0 PL=0
MOVL C00729 V=800.0 PL=0
MOVL C00730 V=800.0 PL=0
MOVL C00731 V=800.0 PL=0
MOVL C00732 V=800.0 PL=0
MOVL C00733 V=800.0 PL=0
MOVL C00734 V=800.0 PL=0
MOVL C00735 V=800.0 PL=0
MOVL C00736 V=800.0 PL=0
MOVL C00737 V=800.0 PL=0
MOVL C00738 V=800.0 PL=0
MOVL C00739 V=800.0 PL=0
MOVL C00740 V=800.0 PL=0
MOVL C00741 V=800.0 PL=0
MOVL C00742 V=800.0 PL=0
MOVL C00743 V=800.0 PL=0
MOVL C00744 V=800.0 PL=0
MOVL C00745 V=800.0 PL=0
MOVL C00746 V=800.0 PL=0
MOVL C00747 V=800.0 PL=0
MOVL C00748 V=800.0 PL=0
MOVL C00749 V=800.0 PL=0
MOVL C00750 V=800.0 PL=0
MOVL C00751 V=800.0 PL=0
MOVL C00752 V=800.0 PL=0
MOVL C00753 V=800.0 PL=0
MOVL C00754 V=800.0 PL=0
MOVL C00755 V=800.0 PL=0
MOVL C00756 V=800.0 PL=0
MOVL C00757 V=800.0 PL=0
MOVL C00758 V=800.0 PL=0
MOVL C00759 V=800.0 PL=0
MOVL C00760 V=800.0 PL=0
MOVL C00761 V=800.0 PL=0
MOVL C00762 V=800.0 PL=0
MOVL C00763 V=800.0 PL=0
MOVL C00764 V=800.0 PL=0
MOVL C00765 V=800.0 PL=0
MOVL C00766 V=800.0 PL=0
MOVL C00767 V=800.0 PL=0
MOVL C00768 V=800.0 PL=0
MOVL C00769 V=800.0 PL=0
MOVL C00770 V=800.0 PL=0
MOVL C00771 V=800.0 PL=0
MOVL C00772 V=800.0 PL=0
MOVL C00773 V=800.0 PL=0
MOVL C00774 V=800.0 PL=0
MOVL C00775 V=800.0 PL=0
MOVL C00776 V=800.0 PL=0
MOVL C00777 V=800.0 PL=0
MOVL C00778 V=800.0 PL=0
MOVL C00779 V=800.0 PL=0
MOVL C00780 V=800.0 PL=0
MOVL C00781 V=800.0 PL=0
MOVL C00782 V=800.0 PL=0
MOVL C00783 V=800.0 PL=0
MOVL C00784 V=800.0 PL=0
MOVL C00785 V=800.0 PL=0
MOVL C00786 V=800.0 PL=0
MOVL C00787 V=800.0 PL=0
MOVL C00788 V=800.0 PL=0
MOVL C00789 V=800.0 PL=0
MOVL C00790 V=800.0 PL=0
MOVL C00791 V=800.0 PL=0
MOVL C00792 V=800.0 PL=0
MOVL C00793 V=800.0 PL=0
MOVL C00794 V=800.0 PL=0
MOVL C00795 V=800.0 PL=0
MOVL C00796 V=800.0 PL=0
MOVL C00797 V=800.0 PL=0
MOVL C00798 V=800.0 PL=0
MOVL C00799 V=800.0 PL=0
MOVL C00800 V=800.0 PL=0
MOVL C00801 V=800.0 PL=0
MOVL C00802 V=800.0 PL=0
MOVL C00803 V=800.0 PL=0
MOVL C00804 V=800.0 PL=0
MOVL C00805 V=800.0 PL=0
MOVL C00806 V=800.0 PL=0
MOVL C00807 V=800.0 PL=0
MOVL C00808 V=800.0 PL=0
MOVL C00809 V=800.0 PL=0
MOVL C00810 V=800.0 PL=0
MOVL C00811 V=800.0 PL=0
MOVL C00812 V=800.0 PL=0
MOVL C00813 V=800.0 PL=0
MOVL C00814 V=800.0 PL=0
MOVL C00815 V=800.0 PL=0
MOVL C00816 V=800.0 PL=0
MOVL C00817 V=800.0 PL=0
MOVL C00818 V=800.0 PL=0
MOVL C00819 V=800.0 PL=0
MOVL C00820 V=800.0 PL=0
MOVL C00821 V=800.0 PL=0
MOVL C00822 V=800.0 PL=0
MOVL C00823 V=800.0 PL=0
MOVL C00824 V=800.0 PL=0
MOVL C00825 V=800.0 PL=0
MOVL C00826 V=800.0 PL=0
MOVL C00827 V=800.0 PL=0
MOVL C00828 V=800.0 PL=0
MOVL C00829 V=800.0 PL=0
MOVL C00830 V=800.0 PL=0
MOVL C00831 V=800.0 PL=0
MOVL C00832 V=800.0 PL=0
MOVL C00833 V=800.0 PL=0
MOVL C00834 V=800.0 PL=0
MOVL C00835 V=800.0 PL=0
MOVL C00836 V=800.0 PL=0
MOVL C00837 V=800.0 PL=0
MOVL C00838 V=800.0 PL=0
MOVL C00839 V=800.0 PL=0
MOVL C00840 V=800.0 PL=0
MOVL C00841 V=800.0 PL=0
MOVL C00842 V=800.0 PL=0
MOVL C00843 V=800.0 PL=0
MOVL C00844 V=800.0 PL=0
MOVL C00845 V=800.0 PL=0
MOVL C00846 V=800.0 PL=0
MOVL C00847 V=800.0 PL=0
MOVL C00848 V=800.0 PL=0
MOVL C00849 V=800.0 PL=0
MOVL C00850 V=800.0 PL=0
MOVL C00851 V=800.0 PL=0
MOVL C00852 V=800.0 PL=0
MOVL C00853 V=800.0 PL=0
MOVL C00854 V=800.0 PL=0
MOVL C00855 V=800.0 PL=0
MOVL C00856 V=800.0 PL=0
MOVL C00857 V=800.0 PL=0
MOVL C00858 V=800.0 PL=0
MOVL C00859 V=800.0 PL=0
MOVL C00860 V=800.0 PL=0
MOVL C00861 V=800.0 PL=0
MOVL C00862 V=800.0 PL=0
MOVL C00863 V=800.0 PL=0
MOVL C00864 V=800.0 PL=0
MOVL C00865 V=800.0 PL=0
MOVL C00866 V=800.0 PL=0
MOVL C00867 V=800.0 PL=0
MOVL C00868 V=800.0 PL=0
MOVL C00869 V=800.0 PL=0
MOVL C00870 V=800.0 PL=0
MOVL C00871 V=800.0 PL=0
MOVL C00872 V=800.0 PL=0
MOVL C00873 V=800.0 PL=0
MOVL C00874 V=800.0 PL=0
MOVL C00875 V=800.0 PL=0
MOVL C00876 V=800.0 PL=0
MOVL C00877 V=800.0 PL=0
MOVL C00878 V=800.0 PL=0
MOVL C00879 V=800.0 PL=0
MOVL C00880 V=800.0 PL=0
MOVL C00881 V=800.0 PL=0
MOVL C00882 V=800.0 PL=0
MOVL C00883 V=800.0 PL=0
MOVL C00884 V=800.0 PL=0
MOVL C00885 V=800.0 PL=0
MOVL C00886 V=800.0 PL=0
MOVL C00887 V=800.0 PL=0
MOVL C00888 V=800.0 PL=0
MOVL C00889 V=800.0 PL=0
MOVL C00890 V=800.0 PL=0
MOVL C00891 V=800.0 PL=0
MOVL C00892 V=800.0 PL=0
MOVL C00893 V=800.0 PL=0
MOVL C00894 V=800.0 PL=0
MOVL C00895 V=800.0 PL=0
MOVL C00896 V=800.0 PL=0
MOVL C00897 V=800.0 PL=0
MOVL C00898 V=800.0 PL=0
MOVL C00899 V=800.0 PL=0
MOVL C00900 V=800.0 PL=0
MOVL C00901 V=800.0 PL=0
MOVL C00902 V=800.0 PL=0
MOVL C00903 V=800.0 PL=0
MOVL C00904 V=800.0 PL=0
MOVL C00905 V=800.0 PL=0
MOVL C00906 V=800.0 PL=0
MOVL C00907 V=800.0 PL=0
MOVL C00908 V=800.0 PL=0
MOVL C00909 V=800.0 PL=0
MOVL C00910 V=800.0 PL=0
MOVL C00911 V=800.0 PL=0
MOVL C00912 V=800.0 PL=0
MOVL C00913 V=800.0 PL=0
MOVL C00914 V=800.0 PL=0
MOVL C00915 V=800.0 PL=0
MOVL C00916 V=800.0 PL=0
MOVL C00917 V=800.0 PL=0
MOVL C00918 V=800.0 PL=0
MOVL C00919 V=800.0 PL=0
MOVL C00920 V=800.0 PL=0
MOVL C00921 V=800.0 PL=0
MOVL C00922 V=800.0 PL=0
MOVL C00923 V=800.0 PL=0
MOVL C00924 V=800.0 PL=0
MOVL C00925 V=800.0 PL=0
MOVL C00926 V=800.0 PL=0
MOVL C00927 V=800.0 PL=0
MOVL C00928 V=800.0 PL=0
MOVL C00929 V=800.0 PL=0
MOVL C00930 V=800.0 PL=0
MOVL C00931 V=800.0 PL=0
MOVL C00932 V=800.0 PL=0
MOVL C00933 V=800.0 PL=0
MOVL C00934 V=800.0 PL=0
MOVL C00935 V=800.0 PL=0
MOVL C00936 V=800.0 PL=0
MOVL C00937 V=800.0 PL=0
MOVL C00938 V=800.0 PL=0
MOVL C00939 V=800.0 PL=0
MOVL C00940 V=800.0 PL=0
MOVL C00941 V=800.0 PL=0
MOVL C00942 V=800.0 PL=0
MOVL C00943 V=800.0 PL=0
MOVL C00944 V=800.0 PL=0
MOVL C00945 V=800.0 PL=0
MOVL C00946 V=800.0 PL=0
MOVL C00947 V=800.0 PL=0
MOVL C00948 V=800.0 PL=0
MOVL C00949 V=800.0 PL=0
MOVL C00950 V=800.0 PL=0
MOVL C00951 V=800.0 PL=0
MOVL C00952 V=800.0 PL=0
MOVL C00953 V=800.0 PL=0
MOVL C00954 V=800.0 PL=0
MOVL C00955 V=800.0 PL=0
MOVL C00956 V=800.0 PL=0
MOVL C00957 V=800.0 PL=0
MOVL C00958 V=800.0 PL=0
MOVL C00959 V=800.0 PL=0
MOVL C00960 V=800.0 PL=0
MOVL C00961 V=800.0 PL=0
MOVL C00962 V=800.0 PL=0
MOVL C00963 V=800.0 PL=0
MOVL C00964 V=800.0 PL=0
MOVL C00965 V=800.0 PL=0
MOVL C00966 V=800.0 PL=0
MOVL C00967 V=800.0 PL=0
MOVL C00968 V=800.0 PL=0
MOVL C00969 V=800.0 PL=0
MOVL C00970 V=800.0 PL=0
MOVL C00971 V=800.0 PL=0
MOVL C00972 V=800.0 PL=0
MOVL C00973 V=800.0 PL=0
MOVL C00974 V=800.0 PL=0
MOVL C00975 V=800.0 PL=0
MOVL C00976 V=800.0 PL=0
MOVL C00977 V=800.0 PL=0
MOVL C00978 V=800.0 PL=0
MOVL C00979 V=800.0 PL=0
MOVL C00980 V=800.0 PL=0
MOVL C00981 V=800.0 PL=0
MOVL C00982 V=800.0 PL=0
MOVL C00983 V=800.0 PL=0
MOVL C00984 V=800.0 PL=0
MOVL C00985 V=800.0 PL=0
MOVL C00986 V=800.0 PL=0
MOVL C00987 V=800.0 PL=0
MOVL C00988 V=800.0 PL=0
MOVL C00989 V=800.0 PL=0
MOVL C00990 V=800.0 PL=0
MOVL C00991 V=800.0 PL=0
MOVL C00992 V=800.0 PL=0
MOVL C00993 V=800.0 PL=0
MOVL C00994 V=800.0 PL=0
MOVL C00995 V=800.0 PL=0
MOVL C00996 V=800.0 PL=0
MOVL C00997 V=800.0 PL=0
MOVL C00998 V=800.0 PL=0
MOVL C00999 V=800.0 PL=0
MOVL C01000 V=800.0 PL=0
MOVL C01001 V=800.0 PL=0
MOVL C01002 V=800.0 PL=0
MOVL C01003 V=800.0 PL=0
MOVL C01004 V=800.0 PL=0
MOVL C01005 V=800.0 PL=0
MOVL C01006 V=800.0 PL=0
MOVL C01007 V=800.0 PL=0
MOVL C01008 V=800.0 PL=0
MOVL C01009 V=800.0 PL=0
MOVL C01010 V=800.0 PL=0
MOVL C01011 V=800.0 PL=0
MOVL C01012 V=800.0 PL=0
MOVL C01013 V=800.0 PL=0
MOVL C01014 V=800.0 PL=0
MOVL C01015 V=800.0 PL=0
MOVL C01016 V=800.0 PL=0
MOVL C01017 V=800.0 PL=0
MOVL C01018 V=800.0 PL=0
MOVL C01019 V=800.0 PL=0
MOVL C01020 V=800.0 PL=0
MOVL C01021 V=800.0 PL=0
MOVL C01022 V=800.0 PL=0
MOVL C01023 V=800.0 PL=0
MOVL C01024 V=800.0 PL=0
MOVL C01025 V=800.0 PL=0
MOVL C01026 V=800.0 PL=0
MOVL C01027 V=800.0 PL=0
MOVL C01028 V=800.0 PL=0
MOVL C01029 V=800.0 PL=0
MOVL C01030 V=800.0 PL=0
MOVL C01031 V=800.0 PL=0
MOVL C01032 V=800.0 PL=0
MOVL C01033 V=800.0 PL=0
MOVL C01034 V=800.0 PL=0
MOVL C01035 V=800.0 PL=0
MOVL C01036 V=800.0 PL=0
MOVL C01037 V=800.0 PL=0
MOVL C01038 V=800.0 PL=0
MOVL C01039 V=800.0 PL=0
MOVL C01040 V=800.0 PL=0
MOVL C01041 V=800.0 PL=0
MOVL C01042 V=800.0 PL=0
MOVL C01043 V=800.0 PL=0
MOVL C01044 V=800.0 PL=0
MOVL C01045 V=800.0 PL=0
MOVL C01046 V=800.0 PL=0
MOVL C01047 V=800.0 PL=0
MOVL C01048 V=800.0 PL=0
MOVL C01049 V=800.0 PL=0
MOVL C01050 V=800.0 PL=0
MOVL C01051 V=800.0 PL=0
MOVL C01052 V=800.0 PL=0
MOVL C01053 V=800.0 PL=0
MOVL C01054 V=800.0 PL=0
MOVL C01055 V=800.0 PL=0
MOVL C01056 V=800.0 PL=0
MOVL C01057 V=800.0 PL=0
MOVL C01058 V=800.0 PL=0
MOVL C01059 V=800.0 PL=0
MOVL C01060 V=800.0 PL=0
MOVL C01061 V=800.0 PL=0
MOVL C01062 V=800.0 PL=0
MOVL C01063 V=800.0 PL=0
MOVL C01064 V=800.0 PL=0
MOVL C01065 V=800.0 PL=0
MOVL C01066 V=800.0 PL=0
MOVL C01067 V=800.0 PL=0
MOVL C01068 V=800.0 PL=0
MOVL C01069 V=800.0 PL=0
MOVL C01070 V=800.0 PL=0
MOVL C01071 V=800.0 PL=0
MOVL C01072 V=800.0 PL=0
MOVL C01073 V=800.0 PL=0
MOVL C01074 V=800.0 PL=0
MOVL C01075 V=800.0 PL=0
MOVL C01076 V=800.0 PL=0
MOVL C01077 V=800.0 PL=0
MOVL C01078 V=800.0 PL=0
MOVL C01079 V=800.0 PL=0
MOVL C01080 V=800.0 PL=0
MOVL C01081 V=800.0 PL=0
MOVL C01082 V=800.0 PL=0
MOVL C01083 V=800.0 PL=0
MOVL C01084 V=800.0 PL=0
MOVL C01085 V=800.0 PL=0
MOVL C01086 V=800.0 PL=0
MOVL C01087 V=800.0 PL=0
MOVL C01088 V=800.0 PL=0
MOVL C01089 V=800.0 PL=0
MOVL C01090 V=800.0 PL=0
MOVL C01091 V=800.0 PL=0
MOVL C01092 V=800.0 PL=0
MOVL C01093 V=800.0 PL=0
MOVL C01094 V=800.0 PL=0
MOVL C01095 V=800.0 PL=0
MOVL C01096 V=800.0 PL=0
MOVL C01097 V=800.0 PL=0
MOVL C01098 V=800.0 PL=0
MOVL C01099 V=800.0 PL=0
MOVL C01100 V=800.0 PL=0
MOVL C01101 V=800.0 PL=0
MOVL C01102 V=800.0 PL=0
MOVL C01103 V=800.0 PL=0
MOVL C01104 V=800.0 PL=0
MOVL C01105 V=800.0 PL=0
MOVL C01106 V=800.0 PL=0
MOVL C01107 V=800.0 PL=0
MOVL C01108 V=800.0 PL=0
MOVL C01109 V=800.0 PL=0
MOVL C01110 V=800.0 PL=0
MOVL C01111 V=800.0 PL=0
MOVL C01112 V=800.0 PL=0
MOVL C01113 V=800.0 PL=0
MOVL C01114 V=800.0 PL=0
MOVL C01115 V=800.0 PL=0
MOVL C01116 V=800.0 PL=0
MOVL C01117 V=800.0 PL=0
MOVL C01118 V=800.0 PL=0
MOVL C01119 V=800.0 PL=0
MOVL C01120 V=800.0 PL=0
MOVL C01121 V=800.0 PL=0
MOVL C01122 V=800.0 PL=0
MOVL C01123 V=800.0 PL=0
MOVL C01124 V=800.0 PL=0
MOVL C01125 V=800.0 PL=0
MOVL C01126 V=800.0 PL=0
MOVL C01127 V=800.0 PL=0
MOVL C01128 V=800.0 PL=0
MOVL C01129 V=800.0 PL=0
MOVL C01130 V=800.0 PL=0
MOVL C01131 V=800.0 PL=0
MOVL C01132 V=800.0 PL=0
MOVL C01133 V=800.0 PL=0
MOVL C01134 V=800.0 PL=0
MOVL C01135 V=800.0 PL=0
MOVL C01136 V=800.0 PL=0
MOVL C01137 V=800.0 PL=0
MOVL C01138 V=800.0 PL=0
MOVL C01139 V=800.0 PL=0
MOVL C01140 V=800.0 PL=0
MOVL C01141 V=800.0 PL=0
MOVL C01142 V=800.0 PL=0
MOVL C01143 V=800.0 PL=0
MOVL C01144 V=800.0 PL=0
MOVL C01145 V=800.0 PL=0
MOVL C01146 V=800.0 PL=0
MOVL C01147 V=800.0 PL=0
MOVL C01148 V=800.0 PL=0
MOVL C01149 V=800.0 PL=0
MOVL C01150 V=800.0 PL=0
MOVL C01151 V=800.0 PL=0
MOVL C01152 V=800.0 PL=0
MOVL C01153 V=800.0 PL=0
MOVL C01154 V=800.0 PL=0
MOVL C01155 V=800.0 PL=0
MOVL C01156 V=800.0 PL=0
MOVL C01157 V=800.0 PL=0
MOVL C01158 V=800.0 PL=0
MOVL C01159 V=800.0 PL=0
MOVL C01160 V=800.0 PL=0
MOVL C01161 V=800.0 PL=0
MOVL C01162 V=800.0 PL=0
MOVL C01163 V=800.0 PL=0
MOVL C01164 V=800.0 PL=0
MOVL C01165 V=800.0 PL=0
MOVL C01166 V=800.0 PL=0
MOVL C01167 V=800.0 PL=0
MOVL C01168 V=800.0 PL=0
MOVL C01169 V=800.0 PL=0
MOVL C01170 V=800.0 PL=0
MOVL C01171 V=800.0 PL=0
MOVL C01172 V=800.0 PL=0
MOVL C01173 V=800.0 PL=0
MOVL C01174 V=800.0 PL=0
MOVL C01175 V=800.0 PL=0
MOVL C01176 V=800.0 PL=0
MOVL C01177 V=800.0 PL=0
MOVL C01178 V=800.0 PL=0
MOVL C01179 V=800.0 PL=0
MOVL C01180 V=800.0 PL=0
MOVL C01181 V=800.0 PL=0
MOVL C01182 V=800.0 PL=0
MOVL C01183 V=800.0 PL=0
MOVL C01184 V=800.0 PL=0
MOVL C01185 V=800.0 PL=0
MOVL C01186 V=800.0 PL=0
MOVL C01187 V=800.0 PL=0
MOVL C01188 V=800.0 PL=0
MOVL C01189 V=800.0 PL=0
MOVL C01190 V=800.0 PL=0
MOVL C01191 V=800.0 PL=0
MOVL C01192 V=800.0 PL=0
MOVL C01193 V=800.0 PL=0
MOVL C01194 V=800.0 PL=0
MOVL C01195 V=800.0 PL=0
MOVL C01196 V=800.0 PL=0
MOVL C01197 V=800.0 PL=0
MOVL C01198 V=800.0 PL=0
MOVL C01199 V=800.0 PL=0
MOVL C01200 V=800.0 PL=0
MOVL C01201 V=800.0 PL=0
MOVL C01202 V=800.0 PL=0
MOVL C01203 V=800.0 PL=0
MOVL C01204 V=800.0 PL=0
MOVL C01205 V=800.0 PL=0
MOVL C01206 V=800.0 PL=0
MOVL C01207 V=800.0 PL=0
MOVL C01208 V=800.0 PL=0
MOVL C01209 V=800.0 PL=0
MOVL C01210 V=800.0 PL=0
MOVL C01211 V=800.0 PL=0
MOVL C01212 V=800.0 PL=0
MOVL C01213 V=800.0 PL=0
MOVL C01214 V=800.0 PL=0
MOVL C01215 V=800.0 PL=0
MOVL C01216 V=800.0 PL=0
MOVL C01217 V=800.0 PL=0
MOVL C01218 V=800.0 PL=0
MOVL C01219 V=800.0 PL=0
MOVL C01220 V=800.0 PL=0
MOVL C01221 V=800.0 PL=0
MOVL C01222 V=800.0 PL=0
MOVL C01223 V=800.0 PL=0
MOVL C01224 V=800.0 PL=0
MOVL C01225 V=800.0 PL=0
MOVL C01226 V=800.0 PL=0
MOVL C01227 V=800.0 PL=0
MOVL C01228 V=800.0 PL=0
MOVL C01229 V=800.0 PL=0
MOVL C01230 V=800.0 PL=0
MOVL C01231 V=800.0 PL=0
MOVL C01232 V=800.0 PL=0
MOVL C01233 V=800.0 PL=0
MOVL C01234 V=800.0 PL=0
MOVL C01235 V=800.0 PL=0
MOVL C01236 V=800.0 PL=0
MOVL C01237 V=800.0 PL=0
MOVL C01238 V=800.0 PL=0
MOVL C01239 V=800.0 PL=0
MOVL C01240 V=800.0 PL=0
MOVL C01241 V=800.0 PL=0
MOVL C01242 V=800.0 PL=0
MOVL C01243 V=800.0 PL=0
MOVL C01244 V=800.0 PL=0
MOVL C01245 V=800.0 PL=0
MOVL C01246 V=800.0 PL=0
MOVL C01247 V=800.0 PL=0
MOVL C01248 V=800.0 PL=0
MOVL C01249 V=800.0 PL=0
MOVL C01250 V=800.0 PL=0
MOVL C01251 V=800.0 PL=0
MOVL C01252 V=800.0 PL=0
MOVL C01253 V=800.0 PL=0
MOVL C01254 V=800.0 PL=0
MOVL C01255 V=800.0 PL=0
MOVL C01256 V=800.0 PL=0
MOVL C01257 V=800.0 PL=0
MOVL C01258 V=800.0 PL=0
MOVL C01259 V=800.0 PL=0
MOVL C01260 V=800.0 PL=0
MOVL C01261 V=800.0 PL=0
MOVL C01262 V=800.0 PL=0
MOVL C01263 V=800.0 PL=0
MOVL C01264 V=800.0 PL=0
MOVL C01265 V=800.0 PL=0
MOVL C01266 V=800.0 PL=0
MOVL C01267 V=800.0 PL=0
MOVL C01268 V=800.0 PL=0
MOVL C01269 V=800.0 PL=0
MOVL C01270 V=800.0 PL=0
MOVL C01271 V=800.0 PL=0
MOVL C01272 V=800.0 PL=0
MOVL C01273 V=800.0 PL=0
MOVL C01274 V=800.0 PL=0
MOVL C01275 V=800.0 PL=0
MOVL C01276 V=800.0 PL=0
MOVL C01277 V=800.0 PL=0
MOVL C01278 V=800.0 PL=0
MOVL C01279 V=800.0 PL=0
MOVL C01280 V=800.0 PL=0
MOVL C01281 V=800.0 PL=0
MOVL C01282 V=800.0 PL=0
MOVL C01283 V=800.0 PL=0
MOVL C01284 V=800.0 PL=0
MOVL C01285 V=800.0 PL=0
MOVL C01286 V=800.0 PL=0
MOVL C01287 V=800.0 PL=0
MOVL C01288 V=800.0 PL=0
MOVL C01289 V=800.0 PL=0
MOVL C01290 V=800.0 PL=0
MOVL C01291 V=800.0 PL=0
MOVL C01292 V=800.0 PL=0
MOVL C01293 V=800.0 PL=0
MOVL C01294 V=800.0 PL=0
MOVL C01295 V=800.0 PL=0
MOVL C01296 V=800.0 PL=0
MOVL C01297 V=800.0 PL=0
MOVL C01298 V=800.0 PL=0
MOVL C01299 V=800.0 PL=0
MOVL C01300 V=800.0 PL=0
MOVL C01301 V=800.0 PL=0
MOVL C01302 V=800.0 PL=0
MOVL C01303 V=800.0 PL=0
MOVL C01304 V=800.0 PL=0
MOVL C01305 V=800.0 PL=0
MOVL C01306 V=800.0 PL=0
MOVL C01307 V=800.0 PL=0
MOVL C01308 V=800.0 PL=0
MOVL C01309 V=800.0 PL=0
MOVL C01310 V=800.0 PL=0
MOVL C01311 V=800.0 PL=0
MOVL C01312 V=800.0 PL=0
MOVL C01313 V=800.0 PL=0
MOVL C01314 V=800.0 PL=0
MOVL C01315 V=800.0 PL=0
MOVL C01316 V=800.0 PL=0
MOVL C01317 V=800.0 PL=0
MOVL C01318 V=800.0 PL=0
MOVL C01319 V=800.0 PL=0
MOVL C01320 V=800.0 PL=0
MOVL C01321 V=800.0 PL=0
MOVL C01322 V=800.0 PL=0
MOVL C01323 V=800.0 PL=0
MOVL C01324 V=800.0 PL=0
MOVL C01325 V=800.0 PL=0
MOVL C01326 V=800.0 PL=0
MOVL C01327 V=800.0 PL=0
MOVL C01328 V=800.0 PL=0
MOVL C01329 V=800.0 PL=0
MOVL C01330 V=800.0 PL=0
MOVL C01331 V=800.0 PL=0
MOVL C01332 V=800.0 PL=0
MOVL C01333 V=800.0 PL=0
MOVL C01334 V=800.0 PL=0
MOVL C01335 V=800.0 PL=0
MOVL C01336 V=800.0 PL=0
MOVL C01337 V=800.0 PL=0
MOVL C01338 V=800.0 PL=0
MOVL C01339 V=800.0 PL=0
MOVL C01340 V=800.0 PL=0
MOVL C01341 V=800.0 PL=0
MOVL C01342 V=800.0 PL=0
MOVL C01343 V=800.0 PL=0
MOVL C01344 V=800.0 PL=0
MOVL C01345 V=800.0 PL=0
MOVL C01346 V=800.0 PL=0
MOVL C01347 V=800.0 PL=0
MOVL C01348 V=800.0 PL=0
MOVL C01349 V=800.0 PL=0
MOVL C01350 V=800.0 PL=0
MOVL C01351 V=800.0 PL=0
MOVL C01352 V=800.0 PL=0
MOVL C01353 V=800.0 PL=0
MOVL C01354 V=800.0 PL=0
MOVL C01355 V=800.0 PL=0
MOVL C01356 V=800.0 PL=0
MOVL C01357 V=800.0 PL=0
MOVL C01358 V=800.0 PL=0
MOVL C01359 V=800.0 PL=0
MOVL C01360 V=800.0 PL=0
MOVL C01361 V=800.0 PL=0
MOVL C01362 V=800.0 PL=0
MOVL C01363 V=800.0 PL=0
MOVL C01364 V=800.0 PL=0
MOVL C01365 V=800.0 PL=0
MOVL C01366 V=800.0 PL=0
MOVL C01367 V=800.0 PL=0
MOVL C01368 V=800.0 PL=0
MOVL C01369 V=800.0 PL=0
MOVL C01370 V=800.0 PL=0
MOVL C01371 V=800.0 PL=0
MOVL C01372 V=800.0 PL=0
MOVL C01373 V=800.0 PL=0
MOVL C01374 V=800.0 PL=0
MOVL C01375 V=800.0 PL=0
MOVL C01376 V=800.0 PL=0
MOVL C01377 V=800.0 PL=0
MOVL C01378 V=800.0 PL=0
MOVL C01379 V=800.0 PL=0
MOVL C01380 V=800.0 PL=0
MOVL C01381 V=800.0 PL=0
MOVL C01382 V=800.0 PL=0
MOVL C01383 V=800.0 PL=0
MOVL C01384 V=800.0 PL=0
MOVL C01385 V=800.0 PL=0
MOVL C01386 V=800.0 PL=0
MOVL C01387 V=800.0 PL=0
MOVL C01388 V=800.0 PL=0
MOVL C01389 V=800.0 PL=0
MOVL C01390 V=800.0 PL=0
MOVL C01391 V=800.0 PL=0
MOVL C01392 V=800.0 PL=0
MOVL C01393 V=800.0 PL=0
MOVL C01394 V=800.0 PL=0
MOVL C01395 V=800.0 PL=0
MOVL C01396 V=800.0 PL=0
MOVL C01397 V=800.0 PL=0
MOVL C01398 V=800.0 PL=0
MOVL C01399 V=800.0 PL=0
MOVL C01400 V=800.0 PL=0
MOVL C01401 V=800.0 PL=0
MOVL C01402 V=800.0 PL=0
MOVL C01403 V=800.0 PL=0
MOVL C01404 V=800.0 PL=0
MOVL C01405 V=800.0 PL=0
MOVL C01406 V=800.0 PL=0
MOVL C01407 V=800.0 PL=0
MOVL C01408 V=800.0 PL=0
MOVL C01409 V=800.0 PL=0
MOVL C01410 V=800.0 PL=0
MOVL C01411 V=800.0 PL=0
MOVL C01412 V=800.0 PL=0
MOVL C01413 V=800.0 PL=0
MOVL C01414 V=800.0 PL=0
MOVL C01415 V=800.0 PL=0
MOVL C01416 V=800.0 PL=0
MOVL C01417 V=800.0 PL=0
MOVL C01418 V=800.0 PL=0
MOVL C01419 V=800.0 PL=0
MOVL C01420 V=800.0 PL=0
MOVL C01421 V=800.0 PL=0
MOVL C01422 V=800.0 PL=0
MOVL C01423 V=800.0 PL=0
MOVL C01424 V=800.0 PL=0
MOVL C01425 V=800.0 PL=0
MOVL C01426 V=800.0 PL=0
MOVL C01427 V=800.0 PL=0
MOVL C01428 V=800.0 PL=0
MOVL C01429 V=800.0 PL=0
MOVL C01430 V=800.0 PL=0
MOVL C01431 V=800.0 PL=0
MOVL C01432 V=800.0 PL=0
MOVL C01433 V=800.0 PL=0
MOVL C01434 V=800.0 PL=0
MOVL C01435 V=800.0 PL=0
MOVL C01436 V=800.0 PL=0
MOVL C01437 V=800.0 PL=0
MOVL C01438 V=800.0 PL=0
MOVL C01439 V=800.0 PL=0
MOVL C01440 V=800.0 PL=0
MOVL C01441 V=800.0 PL=0
MOVL C01442 V=800.0 PL=0
MOVL C01443 V=800.0 PL=0
MOVL C01444 V=800.0 PL=0
MOVL C01445 V=800.0 PL=0
MOVL C01446 V=800.0 PL=0
MOVL C01447 V=800.0 PL=0
MOVL C01448 V=800.0 PL=0
MOVL C01449 V=800.0 PL=0
MOVL C01450 V=800.0 PL=0
MOVL C01451 V=800.0 PL=0
MOVL C01452 V=800.0 PL=0
MOVL C01453 V=800.0 PL=0
MOVL C01454 V=800.0 PL=0
MOVL C01455 V=800.0 PL=0
MOVL C01456 V=800.0 PL=0
MOVL C01457 V=800.0 PL=0
MOVL C01458 V=800.0 PL=0
MOVL C01459 V=800.0 PL=0
MOVL C01460 V=800.0 PL=0
MOVL C01461 V=800.0 PL=0
MOVL C01462 V=800.0 PL=0
MOVL C01463 V=800.0 PL=0
MOVL C01464 V=800.0 PL=0
MOVL C01465 V=800.0 PL=0
MOVL C01466 V=800.0 PL=0
MOVL C01467 V=800.0 PL=0
MOVL C01468 V=800.0 PL=0
MOVL C01469 V=800.0 PL=0
MOVL C01470 V=800.0 PL=0
MOVL C01471 V=800.0 PL=0
MOVL C01472 V=800.0 PL=0
MOVL C01473 V=800.0 PL=0
MOVL C01474 V=800.0 PL=0
MOVL C01475 V=800.0 PL=0
MOVL C01476 V=800.0 PL=0
MOVL C01477 V=800.0 PL=0
MOVL C01478 V=800.0 PL=0
MOVL C01479 V=800.0 PL=0
MOVL C01480 V=800.0 PL=0
MOVL C01481 V=800.0 PL=0
MOVL C01482 V=800.0 PL=0
MOVL C01483 V=800.0 PL=0
MOVL C01484 V=800.0 PL=0
MOVL C01485 V=800.0 PL=0
MOVL C01486 V=800.0 PL=0
MOVL C01487 V=800.0 PL=0
MOVL C01488 V=800.0 PL=0
MOVL C01489 V=800.0 PL=0
MOVL C01490 V=800.0 PL=0
MOVL C01491 V=800.0 PL=0
MOVL C01492 V=800.0 PL=0
MOVL C01493 V=800.0 PL=0
MOVL C01494 V=800.0 PL=0
MOVL C01495 V=800.0 PL=0
MOVL C01496 V=800.0 PL=0
MOVL C01497 V=800.0 PL=0
MOVL C01498 V=800.0 PL=0
MOVL C01499 V=800.0 PL=0
MOVL C01500 V=800.0 PL=0
MOVL C01501 V=800.0 PL=0
MOVL C01502 V=800.0 PL=0
MOVL C01503 V=800.0 PL=0
MOVL C01504 V=800.0 PL=0
MOVL C01505 V=800.0 PL=0
MOVL C01506 V=800.0 PL=0
MOVL C01507 V=800.0 PL=0
MOVL C01508 V=800.0 PL=0
MOVL C01509 V=800.0 PL=0
MOVL C01510 V=800.0 PL=0
MOVL C01511 V=800.0 PL=0
MOVL C01512 V=800.0 PL=0
MOVL C01513 V=800.0 PL=0
MOVL C01514 V=800.0 PL=0
MOVL C01515 V=800.0 PL=0
MOVL C01516 V=800.0 PL=0
MOVL C01517 V=800.0 PL=0
MOVL C01518 V=800.0 PL=0
MOVL C01519 V=800.0 PL=0
MOVL C01520 V=800.0 PL=0
MOVL C01521 V=800.0 PL=0
MOVL C01522 V=800.0 PL=0
MOVL C01523 V=800.0 PL=0
MOVL C01524 V=800.0 PL=0
MOVL C01525 V=800.0 PL=0
MOVL C01526 V=800.0 PL=0
MOVL C01527 V=800.0 PL=0
MOVL C01528 V=800.0 PL=0
MOVL C01529 V=800.0 PL=0
MOVL C01530 V=800.0 PL=0
MOVL C01531 V=800.0 PL=0
MOVL C01532 V=800.0 PL=0
MOVL C01533 V=800.0 PL=0
MOVL C01534 V=800.0 PL=0
MOVL C01535 V=800.0 PL=0
MOVL C01536 V=800.0 PL=0
MOVL C01537 V=800.0 PL=0
MOVL C01538 V=800.0 PL=0
MOVL C01539 V=800.0 PL=0
MOVL C01540 V=800.0 PL=0
MOVL C01541 V=800.0 PL=0
MOVL C01542 V=800.0 PL=0
MOVL C01543 V=800.0 PL=0
MOVL C01544 V=800.0 PL=0
MOVL C01545 V=800.0 PL=0
MOVL C01546 V=800.0 PL=0
MOVL C01547 V=800.0 PL=0
MOVL C01548 V=800.0 PL=0
MOVL C01549 V=800.0 PL=0
MOVL C01550 V=800.0 PL=0
MOVL C01551 V=800.0 PL=0
MOVL C01552 V=800.0 PL=0
MOVL C01553 V=800.0 PL=0
MOVL C01554 V=800.0 PL=0
MOVL C01555 V=800.0 PL=0
MOVL C01556 V=800.0 PL=0
MOVL C01557 V=800.0 PL=0
MOVL C01558 V=800.0 PL=0
MOVL C01559 V=800.0 PL=0
MOVL C01560 V=800.0 PL=0
MOVL C01561 V=800.0 PL=0
MOVL C01562 V=800.0 PL=0
MOVL C01563 V=800.0 PL=0
MOVL C01564 V=800.0 PL=0
MOVL C01565 V=800.0 PL=0
MOVL C01566 V=800.0 PL=0
MOVL C01567 V=800.0 PL=0
MOVL C01568 V=800.0 PL=0
MOVL C01569 V=800.0 PL=0
MOVL C01570 V=800.0 PL=0
MOVL C01571 V=800.0 PL=0
MOVL C01572 V=800.0 PL=0
MOVL C01573 V=800.0 PL=0
MOVL C01574 V=800.0 PL=0
MOVL C01575 V=800.0 PL=0
MOVL C01576 V=800.0 PL=0
MOVL C01577 V=800.0 PL=0
MOVL C01578 V=800.0 PL=0
MOVL C01579 V=800.0 PL=0
MOVL C01580 V=800.0 PL=0
MOVL C01581 V=800.0 PL=0
MOVL C01582 V=800.0 PL=0
MOVL C01583 V=800.0 PL=0
MOVL C01584 V=800.0 PL=0
MOVL C01585 V=800.0 PL=0
MOVL C01586 V=800.0 PL=0
MOVL C01587 V=800.0 PL=0
MOVL C01588 V=800.0 PL=0
MOVL C01589 V=800.0 PL=0
MOVL C01590 V=800.0 PL=0
MOVL C01591 V=800.0 PL=0
MOVL C01592 V=800.0 PL=0
MOVL C01593 V=800.0 PL=0
MOVL C01594 V=800.0 PL=0
MOVL C01595 V=800.0 PL=0
MOVL C01596 V=800.0 PL=0
MOVL C01597 V=800.0 PL=0
MOVL C01598 V=800.0 PL=0
MOVL C01599 V=800.0 PL=0
MOVL C01600 V=800.0 PL=0
MOVL C01601 V=800.0 PL=0
MOVL C01602 V=800.0 PL=0
MOVL C01603 V=800.0 PL=0
MOVL C01604 V=800.0 PL=0
MOVL C01605 V=800.0 PL=0
MOVL C01606 V=800.0 PL=0
MOVL C01607 V=800.0 PL=0
MOVL C01608 V=800.0 PL=0
MOVL C01609 V=800.0 PL=0
MOVL C01610 V=800.0 PL=0
MOVL C01611 V=800.0 PL=0
MOVL C01612 V=800.0 PL=0
MOVL C01613 V=800.0 PL=0
MOVL C01614 V=800.0 PL=0
MOVL C01615 V=800.0 PL=0
MOVL C01616 V=800.0 PL=0
MOVL C01617 V=800.0 PL=0
MOVL C01618 V=800.0 PL=0
MOVL C01619 V=800.0 PL=0
MOVL C01620 V=800.0 PL=0
MOVL C01621 V=800.0 PL=0
MOVL C01622 V=800.0 PL=0
MOVL C01623 V=800.0 PL=0
MOVL C01624 V=800.0 PL=0
MOVL C01625 V=800.0 PL=0
MOVL C01626 V=800.0 PL=0
MOVL C01627 V=800.0 PL=0
MOVL C01628 V=800.0 PL=0
MOVL C01629 V=800.0 PL=0
MOVL C01630 V=800.0 PL=0
MOVL C01631 V=800.0 PL=0
MOVL C01632 V=800.0 PL=0
MOVL C01633 V=800.0 PL=0
MOVL C01634 V=800.0 PL=0
MOVL C01635 V=800.0 PL=0
MOVL C01636 V=800.0 PL=0
MOVL C01637 V=800.0 PL=0
MOVL C01638 V=800.0 PL=0
MOVL C01639 V=800.0 PL=0
MOVL C01640 V=800.0 PL=0
MOVL C01641 V=800.0 PL=0
MOVL C01642 V=800.0 PL=0
MOVL C01643 V=800.0 PL=0
MOVL C01644 V=800.0 PL=0
MOVL C01645 V=800.0 PL=0
MOVL C01646 V=800.0 PL=0
MOVL C01647 V=800.0 PL=0
MOVL C01648 V=800.0 PL=0
MOVL C01649 V=800.0 PL=0
MOVL C01650 V=800.0 PL=0
MOVL C01651 V=800.0 PL=0
MOVL C01652 V=800.0 PL=0
MOVL C01653 V=800.0 PL=0
MOVL C01654 V=800.0 PL=0
MOVL C01655 V=800.0 PL=0
MOVL C01656 V=800.0 PL=0
MOVL C01657 V=800.0 PL=0
MOVL C01658 V=800.0 PL=0
MOVL C01659 V=800.0 PL=0
MOVL C01660 V=800.0 PL=0
MOVL C01661 V=800.0 PL=0
MOVL C01662 V=800.0 PL=0
MOVL C01663 V=800.0 PL=0
MOVL C01664 V=800.0 PL=0
MOVL C01665 V=800.0 PL=0
MOVL C01666 V=800.0 PL=0
MOVL C01667 V=800.0 PL=0
MOVL C01668 V=800.0 PL=0
MOVL C01669 V=800.0 PL=0
MOVL C01670 V=800.0 PL=0
MOVL C01671 V=800.0 PL=0
MOVL C01672 V=800.0 PL=0
MOVL C01673 V=800.0 PL=0
MOVL C01674 V=800.0 PL=0
MOVL C01675 V=800.0 PL=0
MOVL C01676 V=800.0 PL=0
MOVL C01677 V=800.0 PL=0
MOVL C01678 V=800.0 PL=0
MOVL C01679 V=800.0 PL=0
MOVL C01680 V=800.0 PL=0
MOVL C01681 V=800.0 PL=0
MOVL C01682 V=800.0 PL=0
MOVL C01683 V=800.0 PL=0
MOVL C01684 V=800.0 PL=0
MOVL C01685 V=800.0 PL=0
MOVL C01686 V=800.0 PL=0
MOVL C01687 V=800.0 PL=0
MOVL C01688 V=800.0 PL=0
MOVL C01689 V=800.0 PL=0
MOVL C01690 V=800.0 PL=0
MOVL C01691 V=800.0 PL=0
MOVL C01692 V=800.0 PL=0
MOVL C01693 V=800.0 PL=0
MOVL C01694 V=800.0 PL=0
MOVL C01695 V=800.0 PL=0
MOVL C01696 V=800.0 PL=0
MOVL C01697 V=800.0 PL=0
MOVL C01698 V=800.0 PL=0
MOVL C01699 V=800.0 PL=0
MOVL C01700 V=800.0 PL=0
MOVL C01701 V=800.0 PL=0
MOVL C01702 V=800.0 PL=0
MOVL C01703 V=800.0 PL=0
MOVL C01704 V=800.0 PL=0
MOVL C01705 V=800.0 PL=0
MOVL C01706 V=800.0 PL=0
MOVL C01707 V=800.0 PL=0
MOVL C01708 V=800.0 PL=0
MOVL C01709 V=800.0 PL=0
MOVL C01710 V=800.0 PL=0
MOVL C01711 V=800.0 PL=0
MOVL C01712 V=800.0 PL=0
MOVL C01713 V=800.0 PL=0
MOVL C01714 V=800.0 PL=0
MOVL C01715 V=800.0 PL=0
MOVL C01716 V=800.0 PL=0
MOVL C01717 V=800.0 PL=0
MOVL C01718 V=800.0 PL=0
MOVL C01719 V=800.0 PL=0
MOVL C01720 V=800.0 PL=0
MOVL C01721 V=800.0 PL=0
MOVL C01722 V=800.0 PL=0
MOVL C01723 V=800.0 PL=0
MOVL C01724 V=800.0 PL=0
MOVL C01725 V=800.0 PL=0
MOVL C01726 V=800.0 PL=0
MOVL C01727 V=800.0 PL=0
MOVL C01728 V=800.0 PL=0
MOVL C01729 V=800.0 PL=0
MOVL C01730 V=800.0 PL=0
MOVL C01731 V=800.0 PL=0
MOVL C01732 V=800.0 PL=0
MOVL C01733 V=800.0 PL=0
MOVL C01734 V=800.0 PL=0
MOVL C01735 V=800.0 PL=0
MOVL C01736 V=800.0 PL=0
MOVL C01737 V=800.0 PL=0
MOVL C01738 V=800.0 PL=0
MOVL C01739 V=800.0 PL=0
MOVL C01740 V=800.0 PL=0
MOVL C01741 V=800.0 PL=0
MOVL C01742 V=800.0 PL=0
MOVL C01743 V=800.0 PL=0
MOVL C01744 V=800.0 PL=0
MOVL C01745 V=800.0 PL=0
MOVL C01746 V=800.0 PL=0
MOVL C01747 V=800.0 PL=0
MOVL C01748 V=800.0 PL=0
MOVL C01749 V=800.0 PL=0
MOVL C01750 V=800.0 PL=0
MOVL C01751 V=800.0 PL=0
MOVL C01752 V=800.0 PL=0
MOVL C01753 V=800.0 PL=0
MOVL C01754 V=800.0 PL=0
MOVL C01755 V=800.0 PL=0
MOVL C01756 V=800.0 PL=0
MOVL C01757 V=800.0 PL=0
MOVL C01758 V=800.0 PL=0
MOVL C01759 V=800.0 PL=0
MOVL C01760 V=800.0 PL=0
MOVL C01761 V=800.0 PL=0
MOVL C01762 V=800.0 PL=0
MOVL C01763 V=800.0 PL=0
MOVL C01764 V=800.0 PL=0
MOVL C01765 V=800.0 PL=0
MOVL C01766 V=800.0 PL=0
MOVL C01767 V=800.0 PL=0
MOVL C01768 V=800.0 PL=0
MOVL C01769 V=800.0 PL=0
MOVL C01770 V=800.0 PL=0
MOVL C01771 V=800.0 PL=0
MOVL C01772 V=800.0 PL=0
MOVL C01773 V=800.0 PL=0
MOVL C01774 V=800.0 PL=0
MOVL C01775 V=800.0 PL=0
MOVL C01776 V=800.0 PL=0
MOVL C01777 V=800.0 PL=0
MOVL C01778 V=800.0 PL=0
MOVL C01779 V=800.0 PL=0
MOVL C01780 V=800.0 PL=0
MOVL C01781 V=800.0 PL=0
MOVL C01782 V=800.0 PL=0
MOVL C01783 V=800.0 PL=0
MOVL C01784 V=800.0 PL=0
MOVL C01785 V=800.0 PL=0
MOVL C01786 V=800.0 PL=0
MOVL C01787 V=800.0 PL=0
MOVL C01788 V=800.0 PL=0
MOVL C01789 V=800.0 PL=0
MOVL C01790 V=800.0 PL=0
MOVL C01791 V=800.0 PL=0
MOVL C01792 V=800.0 PL=0
MOVL C01793 V=800.0 PL=0
MOVL C01794 V=800.0 PL=0
MOVL C01795 V=800.0 PL=0
MOVL C01796 V=800.0 PL=0
MOVL C01797 V=800.0 PL=0
MOVL C01798 V=800.0 PL=0
MOVL C01799 V=800.0 PL=0
MOVL C01800 V=800.0 PL=0
MOVL C01801 V=800.0 PL=0
MOVL C01802 V=800.0 PL=0
MOVL C01803 V=800.0 PL=0
MOVL C01804 V=800.0 PL=0
MOVL C01805 V=800.0 PL=0
MOVL C01806 V=800.0 PL=0
MOVL C01807 V=800.0 PL=0
MOVL C01808 V=800.0 PL=0
MOVL C01809 V=800.0 PL=0
MOVL C01810 V=800.0 PL=0
MOVL C01811 V=800.0 PL=0
MOVL C01812 V=800.0 PL=0
MOVL C01813 V=800.0 PL=0
MOVL C01814 V=800.0 PL=0
MOVL C01815 V=800.0 PL=0
MOVL C01816 V=800.0 PL=0
MOVL C01817 V=800.0 PL=0
MOVL C01818 V=800.0 PL=0
MOVL C01819 V=800.0 PL=0
MOVL C01820 V=800.0 PL=0
MOVL C01821 V=800.0 PL=0
MOVL C01822 V=800.0 PL=0
MOVL C01823 V=800.0 PL=0
MOVL C01824 V=800.0 PL=0
MOVL C01825 V=800.0 PL=0
MOVL C01826 V=800.0 PL=0
MOVL C01827 V=800.0 PL=0
MOVL C01828 V=800.0 PL=0
MOVL C01829 V=800.0 PL=0
MOVL C01830 V=800.0 PL=0
MOVL C01831 V=800.0 PL=0
MOVL C01832 V=800.0 PL=0
MOVL C01833 V=800.0 PL=0
MOVL C01834 V=800.0 PL=0
MOVL C01835 V=800.0 PL=0
MOVL C01836 V=800.0 PL=0
MOVL C01837 V=800.0 PL=0
MOVL C01838 V=800.0 PL=0
MOVL C01839 V=800.0 PL=0
MOVL C01840 V=800.0 PL=0
MOVL C01841 V=800.0 PL=0
MOVL C01842 V=800.0 PL=0
MOVL C01843 V=800.0 PL=0
MOVL C01844 V=800.0 PL=0
MOVL C01845 V=800.0 PL=0
MOVL C01846 V=800.0 PL=0
MOVL C01847 V=800.0 PL=0
MOVL C01848 V=800.0 PL=0
MOVL C01849 V=800.0 PL=0
MOVL C01850 V=800.0 PL=0
MOVL C01851 V=800.0 PL=0
MOVL C01852 V=800.0 PL=0
MOVL C01853 V=800.0 PL=0
MOVL C01854 V=800.0 PL=0
MOVL C01855 V=800.0 PL=0
MOVL C01856 V=800.0 PL=0
MOVL C01857 V=800.0 PL=0
MOVL C01858 V=800.0 PL=0
MOVL C01859 V=800.0 PL=0
MOVL C01860 V=800.0 PL=0
MOVL C01861 V=800.0 PL=0
MOVL C01862 V=800.0 PL=0
MOVL C01863 V=800.0 PL=0
MOVL C01864 V=800.0 PL=0
MOVL C01865 V=800.0 PL=0
MOVL C01866 V=800.0 PL=0
MOVL C01867 V=800.0 PL=0
MOVL C01868 V=800.0 PL=0
MOVL C01869 V=800.0 PL=0
MOVL C01870 V=800.0 PL=0
MOVL C01871 V=800.0 PL=0
MOVL C01872 V=800.0 PL=0
MOVL C01873 V=800.0 PL=0
MOVL C01874 V=800.0 PL=0
MOVL C01875 V=800.0 PL=0
MOVL C01876 V=800.0 PL=0
MOVL C01877 V=800.0 PL=0
MOVL C01878 V=800.0 PL=0
MOVL C01879 V=800.0 PL=0
MOVL C01880 V=800.0 PL=0
MOVL C01881 V=800.0 PL=0
MOVL C01882 V=800.0 PL=0
MOVL C01883 V=800.0 PL=0
MOVL C01884 V=800.0 PL=0
MOVL C01885 V=800.0 PL=0
MOVL C01886 V=800.0 PL=0
MOVL C01887 V=800.0 PL=0
MOVL C01888 V=800.0 PL=0
MOVL C01889 V=800.0 PL=0
MOVL C01890 V=800.0 PL=0
MOVL C01891 V=800.0 PL=0
MOVL C01892 V=800.0 PL=0
MOVL C01893 V=800.0 PL=0
MOVL C01894 V=800.0 PL=0
MOVL C01895 V=800.0 PL=0
MOVL C01896 V=800.0 PL=0
MOVL C01897 V=800.0 PL=0
MOVL C01898 V=800.0 PL=0
MOVL C01899 V=800.0 PL=0
MOVL C01900 V=800.0 PL=0
MOVL C01901 V=800.0 PL=0
MOVL C01902 V=800.0 PL=0
MOVL C01903 V=800.0 PL=0
MOVL C01904 V=800.0 PL=0
MOVL C01905 V=800.0 PL=0
MOVL C01906 V=800.0 PL=0
MOVL C01907 V=800.0 PL=0
MOVL C01908 V=800.0 PL=0
MOVL C01909 V=800.0 PL=0
MOVL C01910 V=800.0 PL=0
MOVL C01911 V=800.0 PL=0
MOVL C01912 V=800.0 PL=0
MOVL C01913 V=800.0 PL=0
MOVL C01914 V=800.0 PL=0
MOVL C01915 V=800.0 PL=0
MOVL C01916 V=800.0 PL=0
MOVL C01917 V=800.0 PL=0
MOVL C01918 V=800.0 PL=0
MOVL C01919 V=800.0 PL=0
MOVL C01920 V=800.0 PL=0
MOVL C01921 V=800.0 PL=0
MOVL C01922 V=800.0 PL=0
MOVL C01923 V=800.0 PL=0
MOVL C01924 V=800.0 PL=0
MOVL C01925 V=800.0 PL=0
MOVL C01926 V=800.0 PL=0
MOVL C01927 V=800.0 PL=0
MOVL C01928 V=800.0 PL=0
MOVL C01929 V=800.0 PL=0
MOVL C01930 V=800.0 PL=0
MOVL C01931 V=800.0 PL=0
MOVL C01932 V=800.0 PL=0
MOVL C01933 V=800.0 PL=0
MOVL C01934 V=800.0 PL=0
MOVL C01935 V=800.0 PL=0
MOVL C01936 V=800.0 PL=0
MOVL C01937 V=800.0 PL=0
MOVL C01938 V=800.0 PL=0
MOVL C01939 V=800.0 PL=0
MOVL C01940 V=800.0 PL=0
MOVL C01941 V=800.0 PL=0
MOVL C01942 V=800.0 PL=0
MOVL C01943 V=800.0 PL=0
MOVL C01944 V=800.0 PL=0
MOVL C01945 V=800.0 PL=0
MOVL C01946 V=800.0 PL=0
MOVL C01947 V=800.0 PL=0
MOVL C01948 V=800.0 PL=0
MOVL C01949 V=800.0 PL=0
MOVL C01950 V=800.0 PL=0
MOVL C01951 V=800.0 PL=0
MOVL C01952 V=800.0 PL=0
MOVL C01953 V=800.0 PL=0
MOVL C01954 V=800.0 PL=0
MOVL C01955 V=800.0 PL=0
MOVL C01956 V=800.0 PL=0
MOVL C01957 V=800.0 PL=0
MOVL C01958 V=800.0 PL=0
MOVL C01959 V=800.0 PL=0
MOVL C01960 V=800.0 PL=0
MOVL C01961 V=800.0 PL=0
MOVL C01962 V=800.0 PL=0
MOVL C01963 V=800.0 PL=0
MOVL C01964 V=800.0 PL=0
MOVL C01965 V=800.0 PL=0
MOVL C01966 V=800.0 PL=0
MOVL C01967 V=800.0 PL=0
MOVL C01968 V=800.0 PL=0
MOVL C01969 V=800.0 PL=0
MOVL C01970 V=800.0 PL=0
MOVL C01971 V=800.0 PL=0
MOVL C01972 V=800.0 PL=0
MOVL C01973 V=800.0 PL=0
MOVL C01974 V=800.0 PL=0
MOVL C01975 V=800.0 PL=0
MOVL C01976 V=800.0 PL=0
MOVL C01977 V=800.0 PL=0
MOVL C01978 V=800.0 PL=0
MOVL C01979 V=800.0 PL=0
MOVL C01980 V=800.0 PL=0
MOVL C01981 V=800.0 PL=0
MOVL C01982 V=800.0 PL=0
MOVL C01983 V=800.0 PL=0
MOVL C01984 V=800.0 PL=0
MOVL C01985 V=800.0 PL=0
MOVL C01986 V=800.0 PL=0
MOVL C01987 V=800.0 PL=0
MOVL C01988 V=800.0 PL=0
MOVL C01989 V=800.0 PL=0
MOVL C01990 V=800.0 PL=0
MOVL C01991 V=800.0 PL=0
MOVL C01992 V=800.0 PL=0
MOVL C01993 V=800.0 PL=0
MOVL C01994 V=800.0 PL=0
MOVL C01995 V=800.0 PL=0
MOVL C01996 V=800.0 PL=0
MOVL C01997 V=800.0 PL=0
MOVL C01998 V=800.0 PL=0
MOVL C01999 V=800.0 PL=0
MOVL C02000 V=800.0 PL=0
MOVL C02001 V=800.0 PL=0
MOVL C02002 V=800.0 PL=0
MOVL C02003 V=800.0 PL=0
MOVL C02004 V=800.0 PL=0
MOVL C02005 V=800.0 PL=0
MOVL C02006 V=800.0 PL=0
MOVL C02007 V=800.0 PL=0
MOVL C02008 V=800.0 PL=0
MOVL C02009 V=800.0 PL=0
MOVL C02010 V=800.0 PL=0
MOVL C02011 V=800.0 PL=0
MOVL C02012 V=800.0 PL=0
MOVL C02013 V=800.0 PL=0
MOVL C02014 V=800.0 PL=0
MOVL C02015 V=800.0 PL=0
MOVL C02016 V=800.0 PL=0
MOVL C02017 V=800.0 PL=0
MOVL C02018 V=800.0 PL=0
MOVL C02019 V=800.0 PL=0
MOVL C02020 V=800.0 PL=0
MOVL C02021 V=800.0 PL=0
MOVL C02022 V=800.0 PL=0
MOVL C02023 V=800.0 PL=0
MOVL C02024 V=800.0 PL=0
MOVL C02025 V=800.0 PL=0
MOVL C02026 V=800.0 PL=0
MOVL C02027 V=800.0 PL=0
MOVL C02028 V=800.0 PL=0
MOVL C02029 V=800.0 PL=0
MOVL C02030 V=800.0 PL=0
MOVL C02031 V=800.0 PL=0
MOVL C02032 V=800.0 PL=0
MOVL C02033 V=800.0 PL=0
MOVL C02034 V=800.0 PL=0
MOVL C02035 V=800.0 PL=0
MOVL C02036 V=800.0 PL=0
MOVL C02037 V=800.0 PL=0
MOVL C02038 V=800.0 PL=0
MOVL C02039 V=800.0 PL=0
MOVL C02040 V=800.0 PL=0
MOVL C02041 V=800.0 PL=0
MOVL C02042 V=800.0 PL=0
MOVL C02043 V=800.0 PL=0
MOVL C02044 V=800.0 PL=0
MOVL C02045 V=800.0 PL=0
MOVL C02046 V=800.0 PL=0
MOVL C02047 V=800.0 PL=0
MOVL C02048 V=800.0 PL=0
MOVL C02049 V=800.0 PL=0
MOVL C02050 V=800.0 PL=0
MOVL C02051 V=800.0 PL=0
MOVL C02052 V=800.0 PL=0
MOVL C02053 V=800.0 PL=0
MOVL C02054 V=800.0 PL=0
MOVL C02055 V=800.0 PL=0
MOVL C02056 V=800.0 PL=0
MOVL C02057 V=800.0 PL=0
MOVL C02058 V=800.0 PL=0
MOVL C02059 V=800.0 PL=0
MOVL C02060 V=800.0 PL=0
MOVL C02061 V=800.0 PL=0
MOVL C02062 V=800.0 PL=0
MOVL C02063 V=800.0 PL=0
MOVL C02064 V=800.0 PL=0
MOVL C02065 V=800.0 PL=0
MOVL C02066 V=800.0 PL=0
MOVL C02067 V=800.0 PL=0
MOVL C02068 V=800.0 PL=0
MOVL C02069 V=800.0 PL=0
MOVL C02070 V=800.0 PL=0
MOVL C02071 V=800.0 PL=0
MOVL C02072 V=800.0 PL=0
MOVL C02073 V=800.0 PL=0
MOVL C02074 V=800.0 PL=0
MOVL C02075 V=800.0 PL=0
MOVL C02076 V=800.0 PL=0
MOVL C02077 V=800.0 PL=0
MOVL C02078 V=800.0 PL=0
MOVL C02079 V=800.0 PL=0
MOVL C02080 V=800.0 PL=0
MOVL C02081 V=800.0 PL=0
MOVL C02082 V=800.0 PL=0
MOVL C02083 V=800.0 PL=0
MOVL C02084 V=800.0 PL=0
MOVL C02085 V=800.0 PL=0
MOVL C02086 V=800.0 PL=0
MOVL C02087 V=800.0 PL=0
MOVL C02088 V=800.0 PL=0
MOVL C02089 V=800.0 PL=0
MOVL C02090 V=800.0 PL=0
MOVL C02091 V=800.0 PL=0
MOVL C02092 V=800.0 PL=0
MOVL C02093 V=800.0 PL=0
MOVL C02094 V=800.0 PL=0
MOVL C02095 V=800.0 PL=0
MOVL C02096 V=800.0 PL=0
MOVL C02097 V=800.0 PL=0
MOVL C02098 V=800.0 PL=0
MOVL C02099 V=800.0 PL=0
MOVL C02100 V=800.0 PL=0
MOVL C02101 V=800.0 PL=0
MOVL C02102 V=800.0 PL=0
MOVL C02103 V=800.0 PL=0
MOVL C02104 V=800.0 PL=0
MOVL C02105 V=800.0 PL=0
MOVL C02106 V=800.0 PL=0
MOVL C02107 V=800.0 PL=0
MOVL C02108 V=800.0 PL=0
MOVL C02109 V=800.0 PL=0
MOVL C02110 V=800.0 PL=0
MOVL C02111 V=800.0 PL=0
MOVL C02112 V=800.0 PL=0
MOVL C02113 V=800.0 PL=0
MOVL C02114 V=800.0 PL=0
MOVL C02115 V=800.0 PL=0
MOVL C02116 V=800.0 PL=0
MOVL C02117 V=800.0 PL=0
MOVL C02118 V=800.0 PL=0
MOVL C02119 V=800.0 PL=0
MOVL C02120 V=800.0 PL=0
MOVL C02121 V=800.0 PL=0
